LIN {X 0,Y 728.085,Z 811.922,A -85,B 0,C 180,E1 -1269.805,E2 -1269.805} C_VEL
LIN {X 0,Y 728.177,Z 799.737,A -85,B 0,C 180,E1 -1271.003,E2 -1271.003} C_VEL
LIN {X 0,Y 728.297,Z 785.992,A -85,B 0,C 180,E1 -1272.126,E2 -1272.126} C_VEL
LIN {X 0,Y 728.304,Z 784.724,A -85,B 0,C 180,E1 -1272.218,E2 -1272.218} C_VEL
LIN {X 0,Y 727.372,Z 779.122,A -85,B 0,C 180,E1 -1272.633,E2 -1272.633} C_VEL
LIN {X 0,Y 721.623,Z 764.762,A -85,B 0,C 180,E1 -1273.647,E2 -1273.647} C_VEL
LIN {X 0,Y 720.732,Z 758.498,A -85,B 0,C 180,E1 -1274.013,E2 -1274.013} C_VEL
LIN {X 0,Y 720.903,Z 741.804,A -85,B 0,C 180,E1 -1274.819,E2 -1274.819} C_VEL
LIN {X 0,Y 721.108,Z 724.487,A -85,B 0,C 180,E1 -1275.487,E2 -1275.487} C_VEL
LIN {X 0,Y 721.275,Z 705.803,A -85,B 0,C 180,E1 -1276.04,E2 -1276.04} C_VEL
LIN {X 0,Y 721.401,Z 686.903,A -85,B 0,C 180,E1 -1276.439,E2 -1276.439} C_VEL
LIN {X 0,Y 721.479,Z 666.781,A -85,B 0,C 180,E1 -1276.704,E2 -1276.704} C_VEL
LIN {X 0,Y 721.671,Z 473.025,A -85,B 0,C 180,E1 -1278.681,E2 -1278.681} C_VEL
LIN {X 0,Y 721.309,Z 469.724,A -85,B 0,C 180,E1 -1278.739,E2 -1278.739} C_VEL
LIN {X 0,Y 721.774,Z 418.133,A -85,B 0,C 180,E1 -1281.452,E2 -1281.452} C_VEL
LIN {X 0,Y 722.276,Z 363.537,A -85,B 0,C 180,E1 -1284.368,E2 -1284.368} C_VEL
LIN {X 0,Y 722.825,Z 311.685,A -85,B 0,C 180,E1 -1287.193,E2 -1287.193} C_VEL
LIN {X 0,Y 723.408,Z 258.979,A -85,B 0,C 180,E1 -1290.115,E2 -1290.115} C_VEL
LIN {X 0,Y 724.003,Z 208.72,A -85,B 0,C 180,E1 -1292.966,E2 -1292.966} C_VEL
LIN {X 0,Y 723.758,Z 205.468,A -85,B 0,C 180,E1 -1293.167,E2 -1293.167} C_VEL
LIN {X 0,Y 720.196,Z 195.523,A -85,B 0,C 180,E1 -1293.95,E2 -1293.95} C_VEL
LIN {X 0,Y 720.182,Z 195.518,A -85,B 0,C 180,E1 -1296.755,E2 -1296.755} C_VEL
LIN {X 0,Y 720.214,Z 195.521,A -85,B 0,C 180,E1 -1299.599,E2 -1299.599} C_VEL
LIN {X 0,Y 720.16,Z 195.522,A -85,B 0,C 180,E1 -1302.384,E2 -1302.384} C_VEL
LIN {X 0,Y 720.211,Z 195.516,A -85,B 0,C 180,E1 -1305.189,E2 -1305.189} C_VEL
LIN {X 0,Y 720.216,Z 195.521,A -85,B 0,C 180,E1 -1308.211,E2 -1308.211} C_VEL
LIN {X 0,Y 720.148,Z 195.522,A -85,B 0,C 180,E1 -1310.923,E2 -1310.923} C_VEL
LIN {X 0,Y 720.178,Z 195.522,A -85,B 0,C 180,E1 -1314.041,E2 -1314.041} C_VEL
LIN {X 0,Y 720.238,Z 195.651,A -85,B 0,C 180,E1 -1315.596,E2 -1315.596} C_VEL
LIN {X 0,Y 723.958,Z 206.616,A -85,B 0,C 180,E1 -1316.559,E2 -1316.559} C_VEL
LIN {X 0,Y 723.246,Z 247.825,A -85,B 0,C 180,E1 -1319.463,E2 -1319.463} C_VEL
LIN {X 0,Y 722.668,Z 288.727,A -85,B 0,C 180,E1 -1322.252,E2 -1322.252} C_VEL
LIN {X 0,Y 722.544,Z 304.623,A -85,B 0,C 180,E1 -1323.299,E2 -1323.299} C_VEL
LIN {X 0,Y 723.876,Z 312.314,A -85,B 0,C 180,E1 -1323.436,E2 -1323.436} C_VEL
LIN {X 0,Y 722.993,Z 604.896,A -85,B 0,C 180,E1 -1326.562,E2 -1326.562} C_VEL
LIN {X 0,Y 722.818,Z 626.619,A -85,B 0,C 180,E1 -1326.91,E2 -1326.91} C_VEL
LIN {X 0,Y 722.561,Z 650.13,A -85,B 0,C 180,E1 -1327.461,E2 -1327.461} C_VEL
LIN {X 0,Y 722.316,Z 669.51,A -85,B 0,C 180,E1 -1328.052,E2 -1328.052} C_VEL
LIN {X 0,Y 722.014,Z 689.697,A -85,B 0,C 180,E1 -1328.811,E2 -1328.811} C_VEL
LIN {X 0,Y 721.715,Z 710.059,A -85,B 0,C 180,E1 -1329.735,E2 -1329.735} C_VEL
LIN {X 0,Y 721.363,Z 729.936,A -85,B 0,C 180,E1 -1330.822,E2 -1330.822} C_VEL
LIN {X 0,Y 721.062,Z 746.81,A -85,B 0,C 180,E1 -1331.903,E2 -1331.903} C_VEL
LIN {X 0,Y 720.802,Z 763.918,A -85,B 0,C 180,E1 -1333.17,E2 -1333.17} C_VEL
LIN {X 0,Y 720.546,Z 779.819,A -85,B 0,C 180,E1 -1334.548,E2 -1334.548} C_VEL
LIN {X 0,Y 720.356,Z 792.902,A -85,B 0,C 180,E1 -1335.86,E2 -1335.86} C_VEL
LIN {X 0,Y 720.195,Z 806.207,A -85,B 0,C 180,E1 -1337.41,E2 -1337.41} C_VEL
LIN {X 0,Y 720.072,Z 817.974,A -85,B 0,C 180,E1 -1339.035,E2 -1339.035} C_VEL
LIN {X 0,Y 719.998,Z 827.271,A -85,B 0,C 180,E1 -1340.568,E2 -1340.568} C_VEL
LIN {X 0,Y 719.944,Z 835.631,A -85,B 0,C 180,E1 -1342.258,E2 -1342.258} C_VEL
LIN {X 0,Y 719.927,Z 842.505,A -85,B 0,C 180,E1 -1344.021,E2 -1344.021} C_VEL
LIN {X 0,Y 719.92,Z 847.512,A -85,B 0,C 180,E1 -1345.779,E2 -1345.779} C_VEL
LIN {X 0,Y 719.914,Z 850.607,A -85,B 0,C 180,E1 -1347.453,E2 -1347.453} C_VEL
LIN {X 0,Y 719.914,Z 852.289,A -85,B 0,C 180,E1 -1349.204,E2 -1349.204} C_VEL
LIN {X 0,Y 719.909,Z 852.219,A -85,B 0,C 180,E1 -1351.035,E2 -1351.035} C_VEL
LIN {X 0,Y 719.913,Z 850.51,A -85,B 0,C 180,E1 -1352.707,E2 -1352.707} C_VEL
LIN {X 0,Y 719.919,Z 847.147,A -85,B 0,C 180,E1 -1354.461,E2 -1354.461} C_VEL
LIN {X 0,Y 719.936,Z 841.735,A -85,B 0,C 180,E1 -1356.299,E2 -1356.299} C_VEL
LIN {X 0,Y 719.958,Z 834.828,A -85,B 0,C 180,E1 -1358.015,E2 -1358.015} C_VEL
LIN {X 0,Y 720.007,Z 826.408,A -85,B 0,C 180,E1 -1359.674,E2 -1359.674} C_VEL
LIN {X 0,Y 720.103,Z 815.862,A -85,B 0,C 180,E1 -1361.372,E2 -1361.372} C_VEL
LIN {X 0,Y 720.228,Z 804.11,A -85,B 0,C 180,E1 -1362.944,E2 -1362.944} C_VEL
LIN {X 0,Y 720.377,Z 791.433,A -85,B 0,C 180,E1 -1364.386,E2 -1364.386} C_VEL
LIN {X 0,Y 720.595,Z 776.326,A -85,B 0,C 180,E1 -1365.864,E2 -1365.864} C_VEL
LIN {X 0,Y 720.851,Z 759.998,A -85,B 0,C 180,E1 -1367.226,E2 -1367.226} C_VEL
LIN {X 0,Y 721.109,Z 744.471,A -85,B 0,C 180,E1 -1368.346,E2 -1368.346} C_VEL
LIN {X 0,Y 721.411,Z 726.463,A -85,B 0,C 180,E1 -1369.471,E2 -1369.471} C_VEL
LIN {X 0,Y 721.75,Z 706.47,A -85,B 0,C 180,E1 -1370.526,E2 -1370.526} C_VEL
LIN {X 0,Y 722.033,Z 688.563,A -85,B 0,C 180,E1 -1371.325,E2 -1371.325} C_VEL
LIN {X 0,Y 722.331,Z 668.395,A -85,B 0,C 180,E1 -1372.075,E2 -1372.075} C_VEL
LIN {X 0,Y 722.629,Z 645.716,A -85,B 0,C 180,E1 -1372.746,E2 -1372.746} C_VEL
LIN {X 0,Y 722.835,Z 624.224,A -85,B 0,C 180,E1 -1373.224,E2 -1373.224} C_VEL
LIN {X 0,Y 723.001,Z 603.601,A -85,B 0,C 180,E1 -1373.545,E2 -1373.545} C_VEL
LIN {X 0,Y 723.876,Z 312.433,A -85,B 0,C 180,E1 -1376.653,E2 -1376.653} C_VEL
LIN {X 0,Y 722.906,Z 306.324,A -85,B 0,C 180,E1 -1376.758,E2 -1376.758} C_VEL
LIN {X 0,Y 722.485,Z 303.913,A -85,B 0,C 180,E1 -1376.819,E2 -1376.819} C_VEL
LIN {X 0,Y 723.04,Z 261.674,A -85,B 0,C 180,E1 -1379.675,E2 -1379.675} C_VEL
LIN {X 0,Y 723.666,Z 220.838,A -85,B 0,C 180,E1 -1382.512,E2 -1382.512} C_VEL
LIN {X 0,Y 723.746,Z 206.018,A -85,B 0,C 180,E1 -1383.584,E2 -1383.584} C_VEL
LIN {X 0,Y 720.207,Z 195.519,A -85,B 0,C 180,E1 -1384.527,E2 -1384.527} C_VEL
LIN {X 0,Y 720.201,Z 195.524,A -85,B 0,C 180,E1 -1387.452,E2 -1387.452} C_VEL
LIN {X 0,Y 720.212,Z 195.511,A -85,B 0,C 180,E1 -1390.522,E2 -1390.522} C_VEL
LIN {X 0,Y 720.206,Z 195.521,A -85,B 0,C 180,E1 -1393.521,E2 -1393.521} C_VEL
LIN {X 0,Y 720.215,Z 195.509,A -85,B 0,C 180,E1 -1396.589,E2 -1396.589} C_VEL
LIN {X 0,Y 720.219,Z 195.519,A -85,B 0,C 180,E1 -1399.657,E2 -1399.657} C_VEL
LIN {X 0,Y 720.208,Z 195.509,A -85,B 0,C 180,E1 -1402.748,E2 -1402.748} C_VEL
LIN {X 0,Y 720.216,Z 195.521,A -85,B 0,C 180,E1 -1405.695,E2 -1405.695} C_VEL
LIN {X 0,Y 720.211,Z 195.51,A -85,B 0,C 180,E1 -1408.783,E2 -1408.783} C_VEL
LIN {X 0,Y 720.217,Z 195.517,A -85,B 0,C 180,E1 -1411.834,E2 -1411.834} C_VEL
LIN {X 0,Y 720.211,Z 195.51,A -85,B 0,C 180,E1 -1414.86,E2 -1414.86} C_VEL
LIN {X 0,Y 720.212,Z 195.52,A -85,B 0,C 180,E1 -1417.899,E2 -1417.899} C_VEL
LIN {X 0,Y 720.215,Z 195.507,A -85,B 0,C 180,E1 -1420.874,E2 -1420.874} C_VEL
LIN {X 0,Y 720.214,Z 195.52,A -85,B 0,C 180,E1 -1423.888,E2 -1423.888} C_VEL
LIN {X 0,Y 720.219,Z 195.506,A -85,B 0,C 180,E1 -1426.921,E2 -1426.921} C_VEL
LIN {X 0,Y 720.212,Z 195.52,A -85,B 0,C 180,E1 -1429.925,E2 -1429.925} C_VEL
LIN {X 0,Y 720.222,Z 195.506,A -85,B 0,C 180,E1 -1432.902,E2 -1432.902} C_VEL
LIN {X 0,Y 720.211,Z 195.521,A -85,B 0,C 180,E1 -1435.94,E2 -1435.94} C_VEL
LIN {X 0,Y 720.219,Z 195.508,A -85,B 0,C 180,E1 -1438.966,E2 -1438.966} C_VEL
LIN {X 0,Y 720.207,Z 195.52,A -85,B 0,C 180,E1 -1441.989,E2 -1441.989} C_VEL
LIN {X 0,Y 720.21,Z 195.51,A -85,B 0,C 180,E1 -1444.938,E2 -1444.938} C_VEL
LIN {X 0,Y 720.201,Z 195.518,A -85,B 0,C 180,E1 -1448.061,E2 -1448.061} C_VEL
LIN {X 0,Y 720.214,Z 195.51,A -85,B 0,C 180,E1 -1451.046,E2 -1451.046} C_VEL
LIN {X 0,Y 720.202,Z 195.52,A -85,B 0,C 180,E1 -1454.061,E2 -1454.061} C_VEL
LIN {X 0,Y 720.196,Z 195.512,A -85,B 0,C 180,E1 -1456.951,E2 -1456.951} C_VEL
LIN {X 0,Y 720.203,Z 195.521,A -85,B 0,C 180,E1 -1460.055,E2 -1460.055} C_VEL
LIN {X 0,Y 720.184,Z 195.514,A -85,B 0,C 180,E1 -1462.877,E2 -1462.877} C_VEL
LIN {X 0,Y 720.218,Z 195.522,A -85,B 0,C 180,E1 -1465.891,E2 -1465.891} C_VEL
LIN {X 0,Y 720.171,Z 195.516,A -85,B 0,C 180,E1 -1468.711,E2 -1468.711} C_VEL
LIN {X 0,Y 720.219,Z 195.515,A -85,B 0,C 180,E1 -1471.56,E2 -1471.56} C_VEL
LIN {X 0,Y 720.171,Z 195.519,A -85,B 0,C 180,E1 -1474.441,E2 -1474.441} C_VEL
LIN {X 0,Y 720.191,Z 195.514,A -85,B 0,C 180,E1 -1477.163,E2 -1477.163} C_VEL
LIN {X 0,Y 720.188,Z 195.522,A -85,B 0,C 180,E1 -1480.217,E2 -1480.217} C_VEL
LIN {X 0,Y 720.163,Z 195.518,A -85,B 0,C 180,E1 -1482.869,E2 -1482.869} C_VEL
LIN {X 0,Y 720.222,Z 195.518,A -85,B 0,C 180,E1 -1485.756,E2 -1485.756} C_VEL
LIN {X 0,Y 720.158,Z 195.522,A -85,B 0,C 180,E1 -1488.632,E2 -1488.632} C_VEL
LIN {X 0,Y 720.209,Z 195.663,A -85,B 0,C 180,E1 -1490.207,E2 -1490.207} C_VEL
LIN {X 0,Y 721.281,Z 198.701,A -85,B 0,C 180,E1 -1490.423,E2 -1490.423} C_VEL
LIN {X 0,Y 726.57,Z 209.646,A -85,B 0,C 180,E1 -1491.288,E2 -1491.288} C_VEL
LIN {X 0,Y 725.859,Z 260.94,A -85,B 0,C 180,E1 -1493.677,E2 -1493.677} C_VEL
LIN {X 0,Y 725.458,Z 299.229,A -85,B 0,C 180,E1 -1495.402,E2 -1495.402} C_VEL
LIN {X 0,Y 726.47,Z 307.17,A -85,B 0,C 180,E1 -1495.55,E2 -1495.55} C_VEL
LIN {X 0,Y 725.424,Z 570.263,A -85,B 0,C 180,E1 -1498.535,E2 -1498.535} C_VEL
LIN {X 0,Y 724.936,Z 690.96,A -85,B 0,C 180,E1 -1499.899,E2 -1499.899} C_VEL
LIN {X 0,Y 724.634,Z 716.508,A -85,B 0,C 180,E1 -1500.332,E2 -1500.332} C_VEL
LIN {X 0,Y 724.35,Z 738.123,A -85,B 0,C 180,E1 -1500.832,E2 -1500.832} C_VEL
LIN {X 0,Y 724.01,Z 761.286,A -85,B 0,C 180,E1 -1501.501,E2 -1501.501} C_VEL
LIN {X 0,Y 723.566,Z 783.363,A -85,B 0,C 180,E1 -1502.289,E2 -1502.289} C_VEL
LIN {X 0,Y 723.176,Z 805.236,A -85,B 0,C 180,E1 -1503.209,E2 -1503.209} C_VEL
LIN {X 0,Y 722.679,Z 827.148,A -85,B 0,C 180,E1 -1504.294,E2 -1504.294} C_VEL
LIN {X 0,Y 722.248,Z 847.62,A -85,B 0,C 180,E1 -1505.46,E2 -1505.46} C_VEL
LIN {X 0,Y 721.793,Z 867.842,A -85,B 0,C 180,E1 -1506.789,E2 -1506.789} C_VEL
LIN {X 0,Y 721.414,Z 886.71,A -85,B 0,C 180,E1 -1508.195,E2 -1508.195} C_VEL
LIN {X 0,Y 721.029,Z 904.462,A -85,B 0,C 180,E1 -1509.715,E2 -1509.715} C_VEL
LIN {X 0,Y 720.755,Z 920.964,A -85,B 0,C 180,E1 -1511.309,E2 -1511.309} C_VEL
LIN {X 0,Y 720.478,Z 935.22,A -85,B 0,C 180,E1 -1512.889,E2 -1512.889} C_VEL
LIN {X 0,Y 720.304,Z 948.442,A -85,B 0,C 180,E1 -1514.542,E2 -1514.542} C_VEL
LIN {X 0,Y 720.157,Z 960.276,A -85,B 0,C 180,E1 -1516.266,E2 -1516.266} C_VEL
LIN {X 0,Y 720.066,Z 970.03,A -85,B 0,C 180,E1 -1517.896,E2 -1517.896} C_VEL
LIN {X 0,Y 719.982,Z 980.182,A -85,B 0,C 180,E1 -1519.922,E2 -1519.922} C_VEL
LIN {X 0,Y 719.928,Z 986.815,A -85,B 0,C 180,E1 -1521.534,E2 -1521.534} C_VEL
LIN {X 0,Y 719.913,Z 993.245,A -85,B 0,C 180,E1 -1523.46,E2 -1523.46} C_VEL
LIN {X 0,Y 719.916,Z 997.813,A -85,B 0,C 180,E1 -1525.38,E2 -1525.38} C_VEL
LIN {X 0,Y 719.882,Z 1000.685,A -85,B 0,C 180,E1 -1527.134,E2 -1527.134} C_VEL
LIN {X 0,Y 719.891,Z 1002.262,A -85,B 0,C 180,E1 -1529.125,E2 -1529.125} C_VEL
LIN {X 0,Y 719.883,Z 1002.306,A -85,B 0,C 180,E1 -1530.716,E2 -1530.716} C_VEL
LIN {X 0,Y 719.888,Z 1001.017,A -85,B 0,C 180,E1 -1532.627,E2 -1532.627} C_VEL
LIN {X 0,Y 719.917,Z 997.971,A -85,B 0,C 180,E1 -1534.541,E2 -1534.541} C_VEL
LIN {X 0,Y 719.915,Z 993.864,A -85,B 0,C 180,E1 -1536.299,E2 -1536.299} C_VEL
LIN {X 0,Y 719.936,Z 987.422,A -85,B 0,C 180,E1 -1538.305,E2 -1538.305} C_VEL
LIN {X 0,Y 719.968,Z 980.892,A -85,B 0,C 180,E1 -1539.916,E2 -1539.916} C_VEL
LIN {X 0,Y 720.053,Z 971.867,A -85,B 0,C 180,E1 -1541.779,E2 -1541.779} C_VEL
LIN {X 0,Y 720.143,Z 961.081,A -85,B 0,C 180,E1 -1543.608,E2 -1543.608} C_VEL
LIN {X 0,Y 720.295,Z 949.06,A -85,B 0,C 180,E1 -1545.375,E2 -1545.375} C_VEL
LIN {X 0,Y 720.472,Z 935.927,A -85,B 0,C 180,E1 -1547.028,E2 -1547.028} C_VEL
LIN {X 0,Y 720.739,Z 921.74,A -85,B 0,C 180,E1 -1548.607,E2 -1548.607} C_VEL
LIN {X 0,Y 721.008,Z 905.39,A -85,B 0,C 180,E1 -1550.201,E2 -1550.201} C_VEL
LIN {X 0,Y 721.376,Z 888.27,A -85,B 0,C 180,E1 -1551.678,E2 -1551.678} C_VEL
LIN {X 0,Y 721.76,Z 869.107,A -85,B 0,C 180,E1 -1553.121,E2 -1553.121} C_VEL
LIN {X 0,Y 722.231,Z 849.066,A -85,B 0,C 180,E1 -1554.453,E2 -1554.453} C_VEL
LIN {X 0,Y 722.653,Z 827.944,A -85,B 0,C 180,E1 -1555.663,E2 -1555.663} C_VEL
LIN {X 0,Y 723.165,Z 806.229,A -85,B 0,C 180,E1 -1556.747,E2 -1556.747} C_VEL
LIN {X 0,Y 723.547,Z 784.481,A -85,B 0,C 180,E1 -1557.667,E2 -1557.667} C_VEL
LIN {X 0,Y 723.972,Z 762.568,A -85,B 0,C 180,E1 -1558.456,E2 -1558.456} C_VEL
LIN {X 0,Y 724.349,Z 738.334,A -85,B 0,C 180,E1 -1559.162,E2 -1559.162} C_VEL
LIN {X 0,Y 724.63,Z 716.764,A -85,B 0,C 180,E1 -1559.663,E2 -1559.663} C_VEL
LIN {X 0,Y 724.936,Z 691.166,A -85,B 0,C 180,E1 -1560.098,E2 -1560.098} C_VEL
LIN {X 0,Y 725.376,Z 582.637,A -85,B 0,C 180,E1 -1561.326,E2 -1561.326} C_VEL
LIN {X 0,Y 726.451,Z 311.994,A -85,B 0,C 180,E1 -1564.394,E2 -1564.394} C_VEL
LIN {X 0,Y 726.227,Z 304.001,A -85,B 0,C 180,E1 -1564.5,E2 -1564.5} C_VEL
LIN {X 0,Y 725.36,Z 298.429,A -85,B 0,C 180,E1 -1564.618,E2 -1564.618} C_VEL
LIN {X 0,Y 726.223,Z 237.623,A -85,B 0,C 180,E1 -1567.398,E2 -1567.398} C_VEL
LIN {X 0,Y 726.566,Z 209.659,A -85,B 0,C 180,E1 -1568.712,E2 -1568.712} C_VEL
LIN {X 0,Y 721.385,Z 198.876,A -85,B 0,C 180,E1 -1569.587,E2 -1569.587} C_VEL
LIN {X 0,Y 720.172,Z 195.526,A -85,B 0,C 180,E1 -1569.844,E2 -1569.844} C_VEL
LIN {X 0,Y 720.211,Z 195.521,A -85,B 0,C 180,E1 -1572.858,E2 -1572.858} C_VEL
LIN {X 0,Y 720.177,Z 195.524,A -85,B 0,C 180,E1 -1575.704,E2 -1575.704} C_VEL
LIN {X 0,Y 720.221,Z 195.519,A -85,B 0,C 180,E1 -1578.684,E2 -1578.684} C_VEL
LIN {X 0,Y 720.195,Z 195.524,A -85,B 0,C 180,E1 -1581.668,E2 -1581.668} C_VEL
LIN {X 0,Y 720.223,Z 195.521,A -85,B 0,C 180,E1 -1584.625,E2 -1584.625} C_VEL
LIN {X 0,Y 720.201,Z 195.528,A -85,B 0,C 180,E1 -1586.094,E2 -1586.094} C_VEL
LIN {X 0,Y 724.343,Z 207.121,A -85,B 0,C 180,E1 -1587.052,E2 -1587.052} C_VEL
LIN {X 0,Y 723.304,Z 257.17,A -85,B 0,C 180,E1 -1589.926,E2 -1589.926} C_VEL
LIN {X 0,Y 722.6,Z 315.269,A -85,B 0,C 180,E1 -1593.141,E2 -1593.141} C_VEL
LIN {X 0,Y 722.176,Z 369.58,A -85,B 0,C 180,E1 -1596.067,E2 -1596.067} C_VEL
LIN {X 0,Y 721.73,Z 424.416,A -85,B 0,C 180,E1 -1598.972,E2 -1598.972} C_VEL
LIN {X 0,Y 721.364,Z 470.562,A -85,B 0,C 180,E1 -1601.375,E2 -1601.375} C_VEL
LIN {X 0,Y 721.822,Z 478.064,A -85,B 0,C 180,E1 -1601.465,E2 -1601.465} C_VEL
LIN {X 0,Y 721.438,Z 679.938,A -85,B 0,C 180,E1 -1603.541,E2 -1603.541} C_VEL
LIN {X 0,Y 721.316,Z 699.052,A -85,B 0,C 180,E1 -1603.89,E2 -1603.89} C_VEL
LIN {X 0,Y 721.167,Z 717.241,A -85,B 0,C 180,E1 -1604.371,E2 -1604.371} C_VEL
LIN {X 0,Y 720.969,Z 734.998,A -85,B 0,C 180,E1 -1604.992,E2 -1604.992} C_VEL
LIN {X 0,Y 720.803,Z 751.994,A -85,B 0,C 180,E1 -1605.746,E2 -1605.746} C_VEL
LIN {X 0,Y 720.617,Z 767.716,A -85,B 0,C 180,E1 -1606.602,E2 -1606.602} C_VEL
LIN {X 0,Y 720.432,Z 783.102,A -85,B 0,C 180,E1 -1607.618,E2 -1607.618} C_VEL
LIN {X 0,Y 720.274,Z 796.852,A -85,B 0,C 180,E1 -1608.712,E2 -1608.712} C_VEL
LIN {X 0,Y 720.145,Z 809.523,A -85,B 0,C 180,E1 -1609.924,E2 -1609.924} C_VEL
LIN {X 0,Y 720.05,Z 820.643,A -85,B 0,C 180,E1 -1611.214,E2 -1611.214} C_VEL
LIN {X 0,Y 719.983,Z 830.232,A -85,B 0,C 180,E1 -1612.579,E2 -1612.579} C_VEL
LIN {X 0,Y 719.946,Z 837.854,A -85,B 0,C 180,E1 -1613.941,E2 -1613.941} C_VEL
LIN {X 0,Y 719.921,Z 844.045,A -85,B 0,C 180,E1 -1615.379,E2 -1615.379} C_VEL
LIN {X 0,Y 719.914,Z 848.466,A -85,B 0,C 180,E1 -1616.815,E2 -1616.815} C_VEL
LIN {X 0,Y 719.912,Z 851.34,A -85,B 0,C 180,E1 -1618.329,E2 -1618.329} C_VEL
LIN {X 0,Y 719.912,Z 852.449,A -85,B 0,C 180,E1 -1619.841,E2 -1619.841} C_VEL
LIN {X 0,Y 719.913,Z 851.819,A -85,B 0,C 180,E1 -1621.353,E2 -1621.353} C_VEL
LIN {X 0,Y 719.914,Z 849.435,A -85,B 0,C 180,E1 -1622.866,E2 -1622.866} C_VEL
LIN {X 0,Y 719.922,Z 845.232,A -85,B 0,C 180,E1 -1624.381,E2 -1624.381} C_VEL
LIN {X 0,Y 719.936,Z 839.461,A -85,B 0,C 180,E1 -1625.819,E2 -1625.819} C_VEL
LIN {X 0,Y 719.981,Z 831.802,A -85,B 0,C 180,E1 -1627.26,E2 -1627.26} C_VEL
LIN {X 0,Y 720.037,Z 822.605,A -85,B 0,C 180,E1 -1628.626,E2 -1628.626} C_VEL
LIN {X 0,Y 720.131,Z 811.918,A -85,B 0,C 180,E1 -1629.914,E2 -1629.914} C_VEL
LIN {X 0,Y 720.249,Z 799.731,A -85,B 0,C 180,E1 -1631.126,E2 -1631.126} C_VEL
LIN {X 0,Y 720.4,Z 785.987,A -85,B 0,C 180,E1 -1632.261,E2 -1632.261} C_VEL
LIN {X 0,Y 720.572,Z 771.146,A -85,B 0,C 180,E1 -1633.279,E2 -1633.279} C_VEL
LIN {X 0,Y 720.732,Z 758.498,A -85,B 0,C 180,E1 -1634.013,E2 -1634.013} C_VEL
LIN {X 0,Y 719.842,Z 752.168,A -85,B 0,C 180,E1 -1634.364,E2 -1634.364} C_VEL
LIN {X 0,Y 714.42,Z 736.944,A -85,B 0,C 180,E1 -1635.164,E2 -1635.164} C_VEL
LIN {X 0,Y 713.298,Z 730.158,A -85,B 0,C 180,E1 -1635.452,E2 -1635.452} C_VEL
LIN {X 0,Y 713.28,Z 729.152,A -85,B 0,C 180,E1 -1635.489,E2 -1635.489} C_VEL
LIN {X 0,Y 713.505,Z 710.535,A -85,B 0,C 180,E1 -1636.089,E2 -1636.089} C_VEL
LIN {X 0,Y 713.666,Z 691.674,A -85,B 0,C 180,E1 -1636.532,E2 -1636.532} C_VEL
LIN {X 0,Y 713.79,Z 672.625,A -85,B 0,C 180,E1 -1636.823,E2 -1636.823} C_VEL
LIN {X 0,Y 714.094,Z 473.867,A -85,B 0,C 180,E1 -1638.879,E2 -1638.879} C_VEL
LIN {X 0,Y 713.625,Z 469.588,A -85,B 0,C 180,E1 -1638.955,E2 -1638.955} C_VEL
LIN {X 0,Y 714.172,Z 418.046,A -85,B 0,C 180,E1 -1641.692,E2 -1641.692} C_VEL
LIN {X 0,Y 714.783,Z 362.685,A -85,B 0,C 180,E1 -1644.681,E2 -1644.681} C_VEL
LIN {X 0,Y 715.433,Z 312.1,A -85,B 0,C 180,E1 -1647.465,E2 -1647.465} C_VEL
LIN {X 0,Y 716.158,Z 259.687,A -85,B 0,C 180,E1 -1650.401,E2 -1650.401} C_VEL
LIN {X 0,Y 716.883,Z 210.15,A -85,B 0,C 180,E1 -1653.24,E2 -1653.24} C_VEL
LIN {X 0,Y 716.315,Z 207.723,A -85,B 0,C 180,E1 -1653.411,E2 -1653.411} C_VEL
LIN {X 0,Y 712.272,Z 196.512,A -85,B 0,C 180,E1 -1654.307,E2 -1654.307} C_VEL
LIN {X 0,Y 712.274,Z 196.504,A -85,B 0,C 180,E1 -1657.333,E2 -1657.333} C_VEL
LIN {X 0,Y 712.208,Z 196.513,A -85,B 0,C 180,E1 -1660.227,E2 -1660.227} C_VEL
LIN {X 0,Y 712.269,Z 196.511,A -85,B 0,C 180,E1 -1662.91,E2 -1662.91} C_VEL
LIN {X 0,Y 712.265,Z 196.505,A -85,B 0,C 180,E1 -1665.869,E2 -1665.869} C_VEL
LIN {X 0,Y 712.235,Z 196.508,A -85,B 0,C 180,E1 -1668.714,E2 -1668.714} C_VEL
LIN {X 0,Y 712.276,Z 196.512,A -85,B 0,C 180,E1 -1671.566,E2 -1671.566} C_VEL
LIN {X 0,Y 712.234,Z 196.514,A -85,B 0,C 180,E1 -1674.464,E2 -1674.464} C_VEL
LIN {X 0,Y 712.28,Z 196.515,A -85,B 0,C 180,E1 -1675.207,E2 -1675.207} C_VEL
LIN {X 0,Y 716.825,Z 210.095,A -85,B 0,C 180,E1 -1676.417,E2 -1676.417} C_VEL
LIN {X 0,Y 715.958,Z 248.509,A -85,B 0,C 180,E1 -1679.166,E2 -1679.166} C_VEL
LIN {X 0,Y 715.265,Z 289.395,A -85,B 0,C 180,E1 -1681.985,E2 -1681.985} C_VEL
LIN {X 0,Y 715.109,Z 304.617,A -85,B 0,C 180,E1 -1682.999,E2 -1682.999} C_VEL
LIN {X 0,Y 716.715,Z 313.568,A -85,B 0,C 180,E1 -1683.163,E2 -1683.163} C_VEL
LIN {X 0,Y 715.65,Z 604.587,A -85,B 0,C 180,E1 -1686.302,E2 -1686.302} C_VEL
LIN {X 0,Y 715.451,Z 625.147,A -85,B 0,C 180,E1 -1686.631,E2 -1686.631} C_VEL
LIN {X 0,Y 715.193,Z 647.921,A -85,B 0,C 180,E1 -1687.15,E2 -1687.15} C_VEL
LIN {X 0,Y 714.824,Z 669.791,A -85,B 0,C 180,E1 -1687.82,E2 -1687.82} C_VEL
LIN {X 0,Y 714.474,Z 689.691,A -85,B 0,C 180,E1 -1688.576,E2 -1688.576} C_VEL
LIN {X 0,Y 714.107,Z 710.089,A -85,B 0,C 180,E1 -1689.511,E2 -1689.511} C_VEL
LIN {X 0,Y 713.674,Z 729.931,A -85,B 0,C 180,E1 -1690.607,E2 -1690.607} C_VEL
LIN {X 0,Y 713.324,Z 746.817,A -85,B 0,C 180,E1 -1691.7,E2 -1691.7} C_VEL
LIN {X 0,Y 713.005,Z 763.646,A -85,B 0,C 180,E1 -1692.957,E2 -1692.957} C_VEL
LIN {X 0,Y 712.691,Z 779.818,A -85,B 0,C 180,E1 -1694.373,E2 -1694.373} C_VEL
LIN {X 0,Y 712.46,Z 792.9,A -85,B 0,C 180,E1 -1695.7,E2 -1695.7} C_VEL
LIN {X 0,Y 712.265,Z 806.215,A -85,B 0,C 180,E1 -1697.267,E2 -1697.267} C_VEL
LIN {X 0,Y 712.105,Z 818.482,A -85,B 0,C 180,E1 -1698.991,E2 -1698.991} C_VEL
LIN {X 0,Y 712.016,Z 827.705,A -85,B 0,C 180,E1 -1700.543,E2 -1700.543} C_VEL
LIN {X 0,Y 711.958,Z 835.635,A -85,B 0,C 180,E1 -1702.17,E2 -1702.17} C_VEL
LIN {X 0,Y 711.934,Z 842.509,A -85,B 0,C 180,E1 -1703.953,E2 -1703.953} C_VEL
LIN {X 0,Y 711.922,Z 847.507,A -85,B 0,C 180,E1 -1705.731,E2 -1705.731} C_VEL
LIN {X 0,Y 711.915,Z 850.608,A -85,B 0,C 180,E1 -1707.424,E2 -1707.424} C_VEL
LIN {X 0,Y 711.914,Z 852.292,A -85,B 0,C 180,E1 -1709.195,E2 -1709.195} C_VEL
LIN {X 0,Y 711.909,Z 852.214,A -85,B 0,C 180,E1 -1711.046,E2 -1711.046} C_VEL
LIN {X 0,Y 711.912,Z 850.509,A -85,B 0,C 180,E1 -1712.737,E2 -1712.737} C_VEL
LIN {X 0,Y 711.919,Z 847.149,A -85,B 0,C 180,E1 -1714.511,E2 -1714.511} C_VEL
LIN {X 0,Y 711.937,Z 841.731,A -85,B 0,C 180,E1 -1716.37,E2 -1716.37} C_VEL
LIN {X 0,Y 711.97,Z 834.967,A -85,B 0,C 180,E1 -1718.073,E2 -1718.073} C_VEL
LIN {X 0,Y 712.034,Z 826.408,A -85,B 0,C 180,E1 -1719.783,E2 -1719.783} C_VEL
LIN {X 0,Y 712.148,Z 815.858,A -85,B 0,C 180,E1 -1721.5,E2 -1721.5} C_VEL
LIN {X 0,Y 712.297,Z 804.33,A -85,B 0,C 180,E1 -1723.062,E2 -1723.062} C_VEL
LIN {X 0,Y 712.49,Z 791.429,A -85,B 0,C 180,E1 -1724.549,E2 -1724.549} C_VEL
LIN {X 0,Y 712.751,Z 776.122,A -85,B 0,C 180,E1 -1726.062,E2 -1726.062} C_VEL
LIN {X 0,Y 713.054,Z 760.059,A -85,B 0,C 180,E1 -1727.415,E2 -1727.415} C_VEL
LIN {X 0,Y 713.377,Z 744.454,A -85,B 0,C 180,E1 -1728.552,E2 -1728.552} C_VEL
LIN {X 0,Y 713.758,Z 726.057,A -85,B 0,C 180,E1 -1729.712,E2 -1729.712} C_VEL
LIN {X 0,Y 714.156,Z 705.733,A -85,B 0,C 180,E1 -1730.789,E2 -1730.789} C_VEL
LIN {X 0,Y 714.511,Z 687.71,A -85,B 0,C 180,E1 -1731.595,E2 -1731.595} C_VEL
LIN {X 0,Y 714.85,Z 668.384,A -85,B 0,C 180,E1 -1732.319,E2 -1732.319} C_VEL
LIN {X 0,Y 715.217,Z 645.269,A -85,B 0,C 180,E1 -1733.006,E2 -1733.006} C_VEL
LIN {X 0,Y 715.465,Z 624.006,A -85,B 0,C 180,E1 -1733.48,E2 -1733.48} C_VEL
LIN {X 0,Y 715.653,Z 604.059,A -85,B 0,C 180,E1 -1733.794,E2 -1733.794} C_VEL
LIN {X 0,Y 716.712,Z 314.22,A -85,B 0,C 180,E1 -1736.92,E2 -1736.92} C_VEL
LIN {X 0,Y 716.168,Z 309.757,A -85,B 0,C 180,E1 -1736.992,E2 -1736.992} C_VEL
LIN {X 0,Y 715.054,Z 303.905,A -85,B 0,C 180,E1 -1737.12,E2 -1737.12} C_VEL
LIN {X 0,Y 715.713,Z 262.054,A -85,B 0,C 180,E1 -1739.982,E2 -1739.982} C_VEL
LIN {X 0,Y 716.51,Z 225.81,A -85,B 0,C 180,E1 -1742.554,E2 -1742.554} C_VEL
LIN {X 0,Y 716.649,Z 209.27,A -85,B 0,C 180,E1 -1743.74,E2 -1743.74} C_VEL
LIN {X 0,Y 712.244,Z 196.513,A -85,B 0,C 180,E1 -1744.913,E2 -1744.913} C_VEL
LIN {X 0,Y 712.279,Z 196.512,A -85,B 0,C 180,E1 -1747.783,E2 -1747.783} C_VEL
LIN {X 0,Y 712.256,Z 196.503,A -85,B 0,C 180,E1 -1750.752,E2 -1750.752} C_VEL
LIN {X 0,Y 712.28,Z 196.508,A -85,B 0,C 180,E1 -1753.701,E2 -1753.701} C_VEL
LIN {X 0,Y 712.26,Z 196.5,A -85,B 0,C 180,E1 -1756.768,E2 -1756.768} C_VEL
LIN {X 0,Y 712.281,Z 196.507,A -85,B 0,C 180,E1 -1759.778,E2 -1759.778} C_VEL
LIN {X 0,Y 712.268,Z 196.498,A -85,B 0,C 180,E1 -1762.768,E2 -1762.768} C_VEL
LIN {X 0,Y 712.277,Z 196.508,A -85,B 0,C 180,E1 -1765.775,E2 -1765.775} C_VEL
LIN {X 0,Y 712.271,Z 196.5,A -85,B 0,C 180,E1 -1768.801,E2 -1768.801} C_VEL
LIN {X 0,Y 712.276,Z 196.506,A -85,B 0,C 180,E1 -1771.857,E2 -1771.857} C_VEL
LIN {X 0,Y 712.269,Z 196.499,A -85,B 0,C 180,E1 -1774.916,E2 -1774.916} C_VEL
LIN {X 0,Y 712.273,Z 196.509,A -85,B 0,C 180,E1 -1777.9,E2 -1777.9} C_VEL
LIN {X 0,Y 712.274,Z 196.496,A -85,B 0,C 180,E1 -1780.908,E2 -1780.908} C_VEL
LIN {X 0,Y 712.27,Z 196.508,A -85,B 0,C 180,E1 -1783.945,E2 -1783.945} C_VEL
LIN {X 0,Y 712.277,Z 196.495,A -85,B 0,C 180,E1 -1786.965,E2 -1786.965} C_VEL
LIN {X 0,Y 712.268,Z 196.509,A -85,B 0,C 180,E1 -1789.975,E2 -1789.975} C_VEL
LIN {X 0,Y 712.279,Z 196.496,A -85,B 0,C 180,E1 -1792.985,E2 -1792.985} C_VEL
LIN {X 0,Y 712.263,Z 196.508,A -85,B 0,C 180,E1 -1796.056,E2 -1796.056} C_VEL
LIN {X 0,Y 712.282,Z 196.497,A -85,B 0,C 180,E1 -1799.035,E2 -1799.035} C_VEL
LIN {X 0,Y 712.26,Z 196.507,A -85,B 0,C 180,E1 -1802.092,E2 -1802.092} C_VEL
LIN {X 0,Y 712.278,Z 196.499,A -85,B 0,C 180,E1 -1805.074,E2 -1805.074} C_VEL
LIN {X 0,Y 712.262,Z 196.507,A -85,B 0,C 180,E1 -1808.07,E2 -1808.07} C_VEL
LIN {X 0,Y 712.271,Z 196.5,A -85,B 0,C 180,E1 -1811.006,E2 -1811.006} C_VEL
LIN {X 0,Y 712.263,Z 196.509,A -85,B 0,C 180,E1 -1814.06,E2 -1814.06} C_VEL
LIN {X 0,Y 712.261,Z 196.501,A -85,B 0,C 180,E1 -1816.978,E2 -1816.978} C_VEL
LIN {X 0,Y 712.258,Z 196.509,A -85,B 0,C 180,E1 -1820.117,E2 -1820.117} C_VEL
LIN {X 0,Y 712.252,Z 196.503,A -85,B 0,C 180,E1 -1822.971,E2 -1822.971} C_VEL
LIN {X 0,Y 712.265,Z 196.508,A -85,B 0,C 180,E1 -1826.065,E2 -1826.065} C_VEL
LIN {X 0,Y 712.238,Z 196.503,A -85,B 0,C 180,E1 -1828.877,E2 -1828.877} C_VEL
LIN {X 0,Y 712.281,Z 196.508,A -85,B 0,C 180,E1 -1831.865,E2 -1831.865} C_VEL
LIN {X 0,Y 712.228,Z 196.507,A -85,B 0,C 180,E1 -1834.651,E2 -1834.651} C_VEL
LIN {X 0,Y 712.281,Z 196.504,A -85,B 0,C 180,E1 -1837.52,E2 -1837.52} C_VEL
LIN {X 0,Y 712.23,Z 196.51,A -85,B 0,C 180,E1 -1840.456,E2 -1840.456} C_VEL
LIN {X 0,Y 712.251,Z 196.505,A -85,B 0,C 180,E1 -1843.231,E2 -1843.231} C_VEL
LIN {X 0,Y 712.24,Z 196.514,A -85,B 0,C 180,E1 -1846.314,E2 -1846.314} C_VEL
LIN {X 0,Y 712.22,Z 196.51,A -85,B 0,C 180,E1 -1848.929,E2 -1848.929} C_VEL
LIN {X 0,Y 712.307,Z 196.683,A -85,B 0,C 180,E1 -1849.741,E2 -1849.741} C_VEL
LIN {X 0,Y 713.368,Z 199.645,A -85,B 0,C 180,E1 -1849.957,E2 -1849.957} C_VEL
LIN {X 0,Y 719.946,Z 213.509,A -85,B 0,C 180,E1 -1851.055,E2 -1851.055} C_VEL
LIN {X 0,Y 719.057,Z 267.233,A -85,B 0,C 180,E1 -1853.575,E2 -1853.575} C_VEL
LIN {X 0,Y 718.641,Z 299.284,A -85,B 0,C 180,E1 -1855.027,E2 -1855.027} C_VEL
LIN {X 0,Y 719.861,Z 308.443,A -85,B 0,C 180,E1 -1855.203,E2 -1855.203} C_VEL
LIN {X 0,Y 718.584,Z 572.549,A -85,B 0,C 180,E1 -1858.227,E2 -1858.227} C_VEL
LIN {X 0,Y 718.004,Z 691.175,A -85,B 0,C 180,E1 -1859.581,E2 -1859.581} C_VEL
LIN {X 0,Y 717.648,Z 716.767,A -85,B 0,C 180,E1 -1860.019,E2 -1860.019} C_VEL
LIN {X 0,Y 717.298,Z 738.46,A -85,B 0,C 180,E1 -1860.526,E2 -1860.526} C_VEL
LIN {X 0,Y 716.853,Z 762.568,A -85,B 0,C 180,E1 -1861.235,E2 -1861.235} C_VEL
LIN {X 0,Y 716.339,Z 784.486,A -85,B 0,C 180,E1 -1862.031,E2 -1862.031} C_VEL
LIN {X 0,Y 715.831,Z 807.582,A -85,B 0,C 180,E1 -1863.022,E2 -1863.022} C_VEL
LIN {X 0,Y 715.246,Z 828.756,A -85,B 0,C 180,E1 -1864.096,E2 -1864.096} C_VEL
LIN {X 0,Y 714.719,Z 849.755,A -85,B 0,C 180,E1 -1865.317,E2 -1865.317} C_VEL
LIN {X 0,Y 714.182,Z 869.143,A -85,B 0,C 180,E1 -1866.621,E2 -1866.621} C_VEL
LIN {X 0,Y 713.72,Z 887.819,A -85,B 0,C 180,E1 -1868.039,E2 -1868.039} C_VEL
LIN {X 0,Y 713.298,Z 904.462,A -85,B 0,C 180,E1 -1869.485,E2 -1869.485} C_VEL
LIN {X 0,Y 712.937,Z 920.965,A -85,B 0,C 180,E1 -1871.096,E2 -1871.096} C_VEL
LIN {X 0,Y 712.616,Z 935.222,A -85,B 0,C 180,E1 -1872.695,E2 -1872.695} C_VEL
LIN {X 0,Y 712.389,Z 949.06,A -85,B 0,C 180,E1 -1874.45,E2 -1874.45} C_VEL
LIN {X 0,Y 712.21,Z 960.797,A -85,B 0,C 180,E1 -1876.192,E2 -1876.192} C_VEL
LIN {X 0,Y 712.093,Z 970.948,A -85,B 0,C 180,E1 -1877.923,E2 -1877.923} C_VEL
LIN {X 0,Y 711.997,Z 980.538,A -85,B 0,C 180,E1 -1879.89,E2 -1879.89} C_VEL
LIN {X 0,Y 711.935,Z 987.12,A -85,B 0,C 180,E1 -1881.52,E2 -1881.52} C_VEL
LIN {X 0,Y 711.916,Z 993.451,A -85,B 0,C 180,E1 -1883.468,E2 -1883.468} C_VEL
LIN {X 0,Y 711.913,Z 997.814,A -85,B 0,C 180,E1 -1885.327,E2 -1885.327} C_VEL
LIN {X 0,Y 711.882,Z 1000.685,A -85,B 0,C 180,E1 -1887.102,E2 -1887.102} C_VEL
LIN {X 0,Y 711.891,Z 1002.262,A -85,B 0,C 180,E1 -1889.115,E2 -1889.115} C_VEL
LIN {X 0,Y 711.883,Z 1002.306,A -85,B 0,C 180,E1 -1890.724,E2 -1890.724} C_VEL
LIN {X 0,Y 711.887,Z 1001.017,A -85,B 0,C 180,E1 -1892.657,E2 -1892.657} C_VEL
LIN {X 0,Y 711.917,Z 997.972,A -85,B 0,C 180,E1 -1894.592,E2 -1894.592} C_VEL
LIN {X 0,Y 711.915,Z 993.864,A -85,B 0,C 180,E1 -1896.37,E2 -1896.37} C_VEL
LIN {X 0,Y 711.937,Z 987.423,A -85,B 0,C 180,E1 -1898.399,E2 -1898.399} C_VEL
LIN {X 0,Y 711.989,Z 980.892,A -85,B 0,C 180,E1 -1900.029,E2 -1900.029} C_VEL
LIN {X 0,Y 712.085,Z 971.866,A -85,B 0,C 180,E1 -1901.912,E2 -1901.912} C_VEL
LIN {X 0,Y 712.2,Z 961.318,A -85,B 0,C 180,E1 -1903.725,E2 -1903.725} C_VEL
LIN {X 0,Y 712.375,Z 949.642,A -85,B 0,C 180,E1 -1905.467,E2 -1905.467} C_VEL
LIN {X 0,Y 712.602,Z 935.929,A -85,B 0,C 180,E1 -1907.222,E2 -1907.222} C_VEL
LIN {X 0,Y 712.922,Z 921.741,A -85,B 0,C 180,E1 -1908.819,E2 -1908.819} C_VEL
LIN {X 0,Y 713.27,Z 905.39,A -85,B 0,C 180,E1 -1910.43,E2 -1910.43} C_VEL
LIN {X 0,Y 713.688,Z 888.776,A -85,B 0,C 180,E1 -1911.881,E2 -1911.881} C_VEL
LIN {X 0,Y 714.166,Z 869.652,A -85,B 0,C 180,E1 -1913.342,E2 -1913.342} C_VEL
LIN {X 0,Y 714.698,Z 850.418,A -85,B 0,C 180,E1 -1914.64,E2 -1914.64} C_VEL
LIN {X 0,Y 715.218,Z 829.552,A -85,B 0,C 180,E1 -1915.861,E2 -1915.861} C_VEL
LIN {X 0,Y 715.786,Z 808.975,A -85,B 0,C 180,E1 -1916.911,E2 -1916.911} C_VEL
LIN {X 0,Y 716.313,Z 785.727,A -85,B 0,C 180,E1 -1917.92,E2 -1917.92} C_VEL
LIN {X 0,Y 716.771,Z 765.133,A -85,B 0,C 180,E1 -1918.678,E2 -1918.678} C_VEL
LIN {X 0,Y 717.283,Z 740.116,A -85,B 0,C 180,E1 -1919.43,E2 -1919.43} C_VEL
LIN {X 0,Y 717.613,Z 718.69,A -85,B 0,C 180,E1 -1919.94,E2 -1919.94} C_VEL
LIN {X 0,Y 717.992,Z 693.629,A -85,B 0,C 180,E1 -1920.386,E2 -1920.386} C_VEL
LIN {X 0,Y 718.269,Z 642.02,A -85,B 0,C 180,E1 -1920.991,E2 -1920.991} C_VEL
LIN {X 0,Y 719.445,Z 392.284,A -85,B 0,C 180,E1 -1923.827,E2 -1923.827} C_VEL
LIN {X 0,Y 719.68,Z 305.755,A -85,B 0,C 180,E1 -1924.839,E2 -1924.839} C_VEL
LIN {X 0,Y 718.539,Z 298.171,A -85,B 0,C 180,E1 -1925.007,E2 -1925.007} C_VEL
LIN {X 0,Y 719.603,Z 236.709,A -85,B 0,C 180,E1 -1927.846,E2 -1927.846} C_VEL
LIN {X 0,Y 719.965,Z 213.374,A -85,B 0,C 180,E1 -1928.946,E2 -1928.946} C_VEL
LIN {X 0,Y 713.431,Z 199.808,A -85,B 0,C 180,E1 -1930.072,E2 -1930.072} C_VEL
LIN {X 0,Y 712.281,Z 196.511,A -85,B 0,C 180,E1 -1930.336,E2 -1930.336} C_VEL
LIN {X 0,Y 712.279,Z 196.511,A -85,B 0,C 180,E1 -1933.24,E2 -1933.24} C_VEL
LIN {X 0,Y 712.282,Z 196.51,A -85,B 0,C 180,E1 -1936.206,E2 -1936.206} C_VEL
LIN {X 0,Y 712.264,Z 196.512,A -85,B 0,C 180,E1 -1939.171,E2 -1939.171} C_VEL
LIN {X 0,Y 712.28,Z 196.51,A -85,B 0,C 180,E1 -1942.086,E2 -1942.086} C_VEL
LIN {X 0,Y 712.252,Z 196.514,A -85,B 0,C 180,E1 -1945.069,E2 -1945.069} C_VEL
LIN {X 0,Y 712.253,Z 196.683,A -85,B 0,C 180,E1 -1945.655,E2 -1945.655} C_VEL
LIN {X 0,Y 717.389,Z 210.124,A -85,B 0,C 180,E1 -1946.834,E2 -1946.834} C_VEL
LIN {X 0,Y 716.102,Z 258.891,A -85,B 0,C 180,E1 -1949.684,E2 -1949.684} C_VEL
LIN {X 0,Y 715.192,Z 315.897,A -85,B 0,C 180,E1 -1952.885,E2 -1952.885} C_VEL
LIN {X 0,Y 714.624,Z 369.984,A -85,B 0,C 180,E1 -1955.837,E2 -1955.837} C_VEL
LIN {X 0,Y 714.076,Z 424.961,A -85,B 0,C 180,E1 -1958.779,E2 -1958.779} C_VEL
LIN {X 0,Y 713.69,Z 470.224,A -85,B 0,C 180,E1 -1961.147,E2 -1961.147} C_VEL
LIN {X 0,Y 714.267,Z 478.095,A -85,B 0,C 180,E1 -1961.253,E2 -1961.253} C_VEL
LIN {X 0,Y 713.764,Z 680.017,A -85,B 0,C 180,E1 -1963.36,E2 -1963.36} C_VEL
LIN {X 0,Y 713.62,Z 699.074,A -85,B 0,C 180,E1 -1963.712,E2 -1963.712} C_VEL
LIN {X 0,Y 713.437,Z 717.391,A -85,B 0,C 180,E1 -1964.201,E2 -1964.201} C_VEL
LIN {X 0,Y 713.216,Z 734.446,A -85,B 0,C 180,E1 -1964.801,E2 -1964.801} C_VEL
LIN {X 0,Y 713.007,Z 751.19,A -85,B 0,C 180,E1 -1965.545,E2 -1965.545} C_VEL
LIN {X 0,Y 712.784,Z 767.054,A -85,B 0,C 180,E1 -1966.41,E2 -1966.41} C_VEL
LIN {X 0,Y 712.567,Z 781.997,A -85,B 0,C 180,E1 -1967.397,E2 -1967.397} C_VEL
LIN {X 0,Y 712.373,Z 795.932,A -85,B 0,C 180,E1 -1968.503,E2 -1968.503} C_VEL
LIN {X 0,Y 712.209,Z 808.757,A -85,B 0,C 180,E1 -1969.729,E2 -1969.729} C_VEL
LIN {X 0,Y 712.087,Z 820.011,A -85,B 0,C 180,E1 -1971.033,E2 -1971.033} C_VEL
LIN {X 0,Y 712.002,Z 829.721,A -85,B 0,C 180,E1 -1972.414,E2 -1972.414} C_VEL
LIN {X 0,Y 711.952,Z 837.452,A -85,B 0,C 180,E1 -1973.792,E2 -1973.792} C_VEL
LIN {X 0,Y 711.927,Z 843.746,A -85,B 0,C 180,E1 -1975.247,E2 -1975.247} C_VEL
LIN {X 0,Y 711.914,Z 848.468,A -85,B 0,C 180,E1 -1976.779,E2 -1976.779} C_VEL
LIN {X 0,Y 711.913,Z 851.342,A -85,B 0,C 180,E1 -1978.31,E2 -1978.31} C_VEL
LIN {X 0,Y 711.913,Z 852.449,A -85,B 0,C 180,E1 -1979.839,E2 -1979.839} C_VEL
LIN {X 0,Y 711.912,Z 851.818,A -85,B 0,C 180,E1 -1981.368,E2 -1981.368} C_VEL
LIN {X 0,Y 711.915,Z 849.433,A -85,B 0,C 180,E1 -1982.898,E2 -1982.898} C_VEL
LIN {X 0,Y 711.923,Z 845.485,A -85,B 0,C 180,E1 -1984.35,E2 -1984.35} C_VEL
LIN {X 0,Y 711.94,Z 839.812,A -85,B 0,C 180,E1 -1985.804,E2 -1985.804} C_VEL
LIN {X 0,Y 711.987,Z 832.719,A -85,B 0,C 180,E1 -1987.18,E2 -1987.18} C_VEL
LIN {X 0,Y 712.053,Z 823.755,A -85,B 0,C 180,E1 -1988.56,E2 -1988.56} C_VEL
LIN {X 0,Y 712.161,Z 813.333,A -85,B 0,C 180,E1 -1989.863,E2 -1989.863} C_VEL
LIN {X 0,Y 712.307,Z 801.092,A -85,B 0,C 180,E1 -1991.124,E2 -1991.124} C_VEL
LIN {X 0,Y 712.491,Z 787.609,A -85,B 0,C 180,E1 -1992.275,E2 -1992.275} C_VEL
LIN {X 0,Y 712.703,Z 772.501,A -85,B 0,C 180,E1 -1993.343,E2 -1993.343} C_VEL
LIN {X 0,Y 712.932,Z 756.541,A -85,B 0,C 180,E1 -1994.273,E2 -1994.273} C_VEL
LIN {X 0,Y 713.137,Z 739.631,A -85,B 0,C 180,E1 -1995.075,E2 -1995.075} C_VEL
LIN {X 0,Y 713.28,Z 729.152,A -85,B 0,C 180,E1 -1995.489,E2 -1995.489} C_VEL
LIN {X 0,Y 712.665,Z 723.159,A -85,B 0,C 180,E1 -1995.719,E2 -1995.719} C_VEL
LIN {X 0,Y 707.093,Z 705.636,A -85,B 0,C 180,E1 -1996.379,E2 -1996.379} C_VEL
LIN {X 0,Y 705.967,Z 698.377,A -85,B 0,C 180,E1 -1996.579,E2 -1996.579} C_VEL
LIN {X 0,Y 705.952,Z 697.308,A -85,B 0,C 180,E1 -1996.603,E2 -1996.603} C_VEL
LIN {X 0,Y 706.113,Z 677.939,A -85,B 0,C 180,E1 -1996.946,E2 -1996.946} C_VEL
LIN {X 0,Y 706.629,Z 474.731,A -85,B 0,C 180,E1 -1999.105,E2 -1999.105} C_VEL
LIN {X 0,Y 705.964,Z 468.931,A -85,B 0,C 180,E1 -1999.205,E2 -1999.205} C_VEL
LIN {X 0,Y 706.627,Z 415.892,A -85,B 0,C 180,E1 -2002.053,E2 -2002.053} C_VEL
LIN {X 0,Y 707.369,Z 358.655,A -85,B 0,C 180,E1 -2005.181,E2 -2005.181} C_VEL
LIN {X 0,Y 708.094,Z 310.205,A -85,B 0,C 180,E1 -2007.875,E2 -2007.875} C_VEL
LIN {X 0,Y 708.987,Z 256.994,A -85,B 0,C 180,E1 -2010.888,E2 -2010.888} C_VEL
LIN {X 0,Y 709.718,Z 212.196,A -85,B 0,C 180,E1 -2013.484,E2 -2013.484} C_VEL
LIN {X 0,Y 704.332,Z 197.5,A -85,B 0,C 180,E1 -2014.65,E2 -2014.65} C_VEL
LIN {X 0,Y 704.344,Z 197.496,A -85,B 0,C 180,E1 -2017.621,E2 -2017.621} C_VEL
LIN {X 0,Y 704.266,Z 197.502,A -85,B 0,C 180,E1 -2020.454,E2 -2020.454} C_VEL
LIN {X 0,Y 704.345,Z 197.496,A -85,B 0,C 180,E1 -2023.289,E2 -2023.289} C_VEL
LIN {X 0,Y 704.333,Z 197.499,A -85,B 0,C 180,E1 -2026.269,E2 -2026.269} C_VEL
LIN {X 0,Y 704.305,Z 197.495,A -85,B 0,C 180,E1 -2029.174,E2 -2029.174} C_VEL
LIN {X 0,Y 704.268,Z 197.504,A -85,B 0,C 180,E1 -2032.272,E2 -2032.272} C_VEL
LIN {X 0,Y 704.339,Z 197.652,A -85,B 0,C 180,E1 -2034.818,E2 -2034.818} C_VEL
LIN {X 0,Y 709.779,Z 213.038,A -85,B 0,C 180,E1 -2036.218,E2 -2036.218} C_VEL
LIN {X 0,Y 708.933,Z 248.718,A -85,B 0,C 180,E1 -2038.78,E2 -2038.78} C_VEL
LIN {X 0,Y 708.094,Z 278.852,A -85,B 0,C 180,E1 -2040.938,E2 -2040.938} C_VEL
LIN {X 0,Y 707.707,Z 304.681,A -85,B 0,C 180,E1 -2042.693,E2 -2042.693} C_VEL
LIN {X 0,Y 709.572,Z 314.84,A -85,B 0,C 180,E1 -2042.884,E2 -2042.884} C_VEL
LIN {X 0,Y 708.323,Z 604.176,A -85,B 0,C 180,E1 -2046.037,E2 -2046.037} C_VEL
LIN {X 0,Y 708.111,Z 623.549,A -85,B 0,C 180,E1 -2046.344,E2 -2046.344} C_VEL
LIN {X 0,Y 707.825,Z 644.177,A -85,B 0,C 180,E1 -2046.802,E2 -2046.802} C_VEL
LIN {X 0,Y 707.416,Z 667.036,A -85,B 0,C 180,E1 -2047.478,E2 -2047.478} C_VEL
LIN {X 0,Y 707.008,Z 686.572,A -85,B 0,C 180,E1 -2048.208,E2 -2048.208} C_VEL
LIN {X 0,Y 706.609,Z 704.141,A -85,B 0,C 180,E1 -2048.992,E2 -2048.992} C_VEL
LIN {X 0,Y 706.199,Z 722.741,A -85,B 0,C 180,E1 -2049.962,E2 -2049.962} C_VEL
LIN {X 0,Y 705.716,Z 742.117,A -85,B 0,C 180,E1 -2051.166,E2 -2051.166} C_VEL
LIN {X 0,Y 705.32,Z 758.277,A -85,B 0,C 180,E1 -2052.339,E2 -2052.339} C_VEL
LIN {X 0,Y 704.961,Z 774.409,A -85,B 0,C 180,E1 -2053.69,E2 -2053.69} C_VEL
LIN {X 0,Y 704.623,Z 790.595,A -85,B 0,C 180,E1 -2055.285,E2 -2055.285} C_VEL
LIN {X 0,Y 704.384,Z 802.926,A -85,B 0,C 180,E1 -2056.705,E2 -2056.705} C_VEL
LIN {X 0,Y 704.202,Z 814.074,A -85,B 0,C 180,E1 -2058.202,E2 -2058.202} C_VEL
LIN {X 0,Y 704.077,Z 824.984,A -85,B 0,C 180,E1 -2059.94,E2 -2059.94} C_VEL
LIN {X 0,Y 703.991,Z 833.448,A -85,B 0,C 180,E1 -2061.588,E2 -2061.588} C_VEL
LIN {X 0,Y 703.935,Z 839.935,A -85,B 0,C 180,E1 -2063.162,E2 -2063.162} C_VEL
LIN {X 0,Y 703.916,Z 845.471,A -85,B 0,C 180,E1 -2064.866,E2 -2064.866} C_VEL
LIN {X 0,Y 703.903,Z 849.66,A -85,B 0,C 180,E1 -2066.743,E2 -2066.743} C_VEL
LIN {X 0,Y 703.9,Z 851.844,A -85,B 0,C 180,E1 -2068.535,E2 -2068.535} C_VEL
LIN {X 0,Y 703.902,Z 852.452,A -85,B 0,C 180,E1 -2070.326,E2 -2070.326} C_VEL
LIN {X 0,Y 703.911,Z 851.29,A -85,B 0,C 180,E1 -2072.198,E2 -2072.198} C_VEL
LIN {X 0,Y 703.919,Z 848.414,A -85,B 0,C 180,E1 -2073.991,E2 -2073.991} C_VEL
LIN {X 0,Y 703.925,Z 843.802,A -85,B 0,C 180,E1 -2075.788,E2 -2075.788} C_VEL
LIN {X 0,Y 703.954,Z 837.441,A -85,B 0,C 180,E1 -2077.591,E2 -2077.591} C_VEL
LIN {X 0,Y 704.021,Z 829.494,A -85,B 0,C 180,E1 -2079.318,E2 -2079.318} C_VEL
LIN {X 0,Y 704.122,Z 820.083,A -85,B 0,C 180,E1 -2080.969,E2 -2080.969} C_VEL
LIN {X 0,Y 704.287,Z 809.445,A -85,B 0,C 180,E1 -2082.546,E2 -2082.546} C_VEL
LIN {X 0,Y 704.516,Z 795.925,A -85,B 0,C 180,E1 -2084.22,E2 -2084.22} C_VEL
LIN {X 0,Y 704.779,Z 782.443,A -85,B 0,C 180,E1 -2085.638,E2 -2085.638} C_VEL
LIN {X 0,Y 705.124,Z 767.259,A -85,B 0,C 180,E1 -2087.027,E2 -2087.027} C_VEL
LIN {X 0,Y 705.535,Z 749.3,A -85,B 0,C 180,E1 -2088.423,E2 -2088.423} C_VEL
LIN {X 0,Y 705.94,Z 732.752,A -85,B 0,C 180,E1 -2089.528,E2 -2089.528} C_VEL
LIN {X 0,Y 706.371,Z 714.967,A -85,B 0,C 180,E1 -2090.552,E2 -2090.552} C_VEL
LIN {X 0,Y 706.858,Z 693.799,A -85,B 0,C 180,E1 -2091.579,E2 -2091.579} C_VEL
LIN {X 0,Y 707.285,Z 673.767,A -85,B 0,C 180,E1 -2092.376,E2 -2092.376} C_VEL
LIN {X 0,Y 707.599,Z 655.35,A -85,B 0,C 180,E1 -2092.977,E2 -2092.977} C_VEL
LIN {X 0,Y 707.945,Z 636.235,A -85,B 0,C 180,E1 -2093.48,E2 -2093.48} C_VEL
LIN {X 0,Y 708.226,Z 614.339,A -85,B 0,C 180,E1 -2093.912,E2 -2093.912} C_VEL
LIN {X 0,Y 708.439,Z 584.242,A -85,B 0,C 180,E1 -2094.283,E2 -2094.283} C_VEL
LIN {X 0,Y 709.568,Z 313.73,A -85,B 0,C 180,E1 -2097.218,E2 -2097.218} C_VEL
LIN {X 0,Y 707.643,Z 303.896,A -85,B 0,C 180,E1 -2097.428,E2 -2097.428} C_VEL
LIN {X 0,Y 708.447,Z 263.895,A -85,B 0,C 180,E1 -2100.209,E2 -2100.209} C_VEL
LIN {X 0,Y 709.423,Z 230.579,A -85,B 0,C 180,E1 -2102.623,E2 -2102.623} C_VEL
LIN {X 0,Y 709.669,Z 212.635,A -85,B 0,C 180,E1 -2103.914,E2 -2103.914} C_VEL
LIN {X 0,Y 704.312,Z 197.503,A -85,B 0,C 180,E1 -2105.296,E2 -2105.296} C_VEL
LIN {X 0,Y 704.342,Z 197.493,A -85,B 0,C 180,E1 -2108.343,E2 -2108.343} C_VEL
LIN {X 0,Y 704.315,Z 197.496,A -85,B 0,C 180,E1 -2111.322,E2 -2111.322} C_VEL
LIN {X 0,Y 704.337,Z 197.493,A -85,B 0,C 180,E1 -2114.316,E2 -2114.316} C_VEL
LIN {X 0,Y 704.312,Z 197.494,A -85,B 0,C 180,E1 -2117.265,E2 -2117.265} C_VEL
LIN {X 0,Y 704.329,Z 197.494,A -85,B 0,C 180,E1 -2120.177,E2 -2120.177} C_VEL
LIN {X 0,Y 704.314,Z 197.491,A -85,B 0,C 180,E1 -2123.093,E2 -2123.093} C_VEL
LIN {X 0,Y 704.33,Z 197.492,A -85,B 0,C 180,E1 -2126.003,E2 -2126.003} C_VEL
LIN {X 0,Y 704.321,Z 197.491,A -85,B 0,C 180,E1 -2128.98,E2 -2128.98} C_VEL
LIN {X 0,Y 704.336,Z 197.494,A -85,B 0,C 180,E1 -2131.88,E2 -2131.88} C_VEL
LIN {X 0,Y 704.331,Z 197.488,A -85,B 0,C 180,E1 -2134.921,E2 -2134.921} C_VEL
LIN {X 0,Y 704.335,Z 197.498,A -85,B 0,C 180,E1 -2137.901,E2 -2137.901} C_VEL
LIN {X 0,Y 704.334,Z 197.485,A -85,B 0,C 180,E1 -2140.943,E2 -2140.943} C_VEL
LIN {X 0,Y 704.331,Z 197.497,A -85,B 0,C 180,E1 -2143.964,E2 -2143.964} C_VEL
LIN {X 0,Y 704.339,Z 197.483,A -85,B 0,C 180,E1 -2146.955,E2 -2146.955} C_VEL
LIN {X 0,Y 704.326,Z 197.497,A -85,B 0,C 180,E1 -2150.026,E2 -2150.026} C_VEL
LIN {X 0,Y 704.34,Z 197.484,A -85,B 0,C 180,E1 -2152.987,E2 -2152.987} C_VEL
LIN {X 0,Y 704.327,Z 197.498,A -85,B 0,C 180,E1 -2156.011,E2 -2156.011} C_VEL
LIN {X 0,Y 704.342,Z 197.486,A -85,B 0,C 180,E1 -2159.024,E2 -2159.024} C_VEL
LIN {X 0,Y 704.326,Z 197.497,A -85,B 0,C 180,E1 -2162.034,E2 -2162.034} C_VEL
LIN {X 0,Y 704.338,Z 197.488,A -85,B 0,C 180,E1 -2165.05,E2 -2165.05} C_VEL
LIN {X 0,Y 704.322,Z 197.495,A -85,B 0,C 180,E1 -2168.079,E2 -2168.079} C_VEL
LIN {X 0,Y 704.335,Z 197.489,A -85,B 0,C 180,E1 -2171.049,E2 -2171.049} C_VEL
LIN {X 0,Y 704.317,Z 197.497,A -85,B 0,C 180,E1 -2174.157,E2 -2174.157} C_VEL
LIN {X 0,Y 704.333,Z 197.49,A -85,B 0,C 180,E1 -2177.089,E2 -2177.089} C_VEL
LIN {X 0,Y 704.315,Z 197.497,A -85,B 0,C 180,E1 -2180.181,E2 -2180.181} C_VEL
LIN {X 0,Y 704.324,Z 197.491,A -85,B 0,C 180,E1 -2183.084,E2 -2183.084} C_VEL
LIN {X 0,Y 704.313,Z 197.496,A -85,B 0,C 180,E1 -2186.204,E2 -2186.204} C_VEL
LIN {X 0,Y 704.314,Z 197.491,A -85,B 0,C 180,E1 -2189.047,E2 -2189.047} C_VEL
LIN {X 0,Y 704.311,Z 197.499,A -85,B 0,C 180,E1 -2192.207,E2 -2192.207} C_VEL
LIN {X 0,Y 704.301,Z 197.494,A -85,B 0,C 180,E1 -2194.999,E2 -2194.999} C_VEL
LIN {X 0,Y 704.332,Z 197.497,A -85,B 0,C 180,E1 -2198.034,E2 -2198.034} C_VEL
LIN {X 0,Y 704.286,Z 197.496,A -85,B 0,C 180,E1 -2200.825,E2 -2200.825} C_VEL
LIN {X 0,Y 704.345,Z 197.495,A -85,B 0,C 180,E1 -2203.737,E2 -2203.737} C_VEL
LIN {X 0,Y 704.283,Z 197.501,A -85,B 0,C 180,E1 -2206.628,E2 -2206.628} C_VEL
LIN {X 0,Y 704.318,Z 197.608,A -85,B 0,C 180,E1 -2209.236,E2 -2209.236} C_VEL
LIN {X 0,Y 705.292,Z 200.424,A -85,B 0,C 180,E1 -2209.454,E2 -2209.454} C_VEL
LIN {X 0,Y 706.704,Z 203.245,A -85,B 0,C 180,E1 -2209.695,E2 -2209.695} C_VEL
LIN {X 0,Y 713.285,Z 217.385,A -85,B 0,C 180,E1 -2210.824,E2 -2210.824} C_VEL
LIN {X 0,Y 712.298,Z 270.275,A -85,B 0,C 180,E1 -2213.318,E2 -2213.318} C_VEL
LIN {X 0,Y 711.848,Z 299.334,A -85,B 0,C 180,E1 -2214.644,E2 -2214.644} C_VEL
LIN {X 0,Y 713.279,Z 309.701,A -85,B 0,C 180,E1 -2214.85,E2 -2214.85} C_VEL
LIN {X 0,Y 711.768,Z 574.626,A -85,B 0,C 180,E1 -2217.911,E2 -2217.911} C_VEL
LIN {X 0,Y 711.095,Z 691.218,A -85,B 0,C 180,E1 -2219.254,E2 -2219.254} C_VEL
LIN {X 0,Y 710.694,Z 716.763,A -85,B 0,C 180,E1 -2219.695,E2 -2219.695} C_VEL
LIN {X 0,Y 710.27,Z 738.453,A -85,B 0,C 180,E1 -2220.205,E2 -2220.205} C_VEL
LIN {X 0,Y 709.758,Z 762.564,A -85,B 0,C 180,E1 -2220.92,E2 -2220.92} C_VEL
LIN {X 0,Y 709.159,Z 784.49,A -85,B 0,C 180,E1 -2221.722,E2 -2221.722} C_VEL
LIN {X 0,Y 708.561,Z 807.17,A -85,B 0,C 180,E1 -2222.702,E2 -2222.702} C_VEL
LIN {X 0,Y 707.877,Z 828.76,A -85,B 0,C 180,E1 -2223.806,E2 -2223.806} C_VEL
LIN {X 0,Y 707.237,Z 849.752,A -85,B 0,C 180,E1 -2225.038,E2 -2225.038} C_VEL
LIN {X 0,Y 706.624,Z 869.053,A -85,B 0,C 180,E1 -2226.349,E2 -2226.349} C_VEL
LIN {X 0,Y 706.064,Z 887.763,A -85,B 0,C 180,E1 -2227.783,E2 -2227.783} C_VEL
LIN {X 0,Y 705.564,Z 904.786,A -85,B 0,C 180,E1 -2229.281,E2 -2229.281} C_VEL
LIN {X 0,Y 705.127,Z 920.967,A -85,B 0,C 180,E1 -2230.879,E2 -2230.879} C_VEL
LIN {X 0,Y 704.764,Z 935.224,A -85,B 0,C 180,E1 -2232.496,E2 -2232.496} C_VEL
LIN {X 0,Y 704.49,Z 949.061,A -85,B 0,C 180,E1 -2234.271,E2 -2234.271} C_VEL
LIN {X 0,Y 704.274,Z 960.798,A -85,B 0,C 180,E1 -2236.033,E2 -2236.033} C_VEL
LIN {X 0,Y 704.126,Z 971.406,A -85,B 0,C 180,E1 -2237.868,E2 -2237.868} C_VEL
LIN {X 0,Y 704.018,Z 980.722,A -85,B 0,C 180,E1 -2239.817,E2 -2239.817} C_VEL
LIN {X 0,Y 703.942,Z 987.424,A -85,B 0,C 180,E1 -2241.505,E2 -2241.505} C_VEL
LIN {X 0,Y 703.916,Z 993.864,A -85,B 0,C 180,E1 -2243.557,E2 -2243.557} C_VEL
LIN {X 0,Y 703.915,Z 997.973,A -85,B 0,C 180,E1 -2245.356,E2 -2245.356} C_VEL
LIN {X 0,Y 703.884,Z 1000.91,A -85,B 0,C 180,E1 -2247.232,E2 -2247.232} C_VEL
LIN {X 0,Y 703.888,Z 1002.284,A -85,B 0,C 180,E1 -2249.186,E2 -2249.186} C_VEL
LIN {X 0,Y 703.888,Z 1002.284,A -85,B 0,C 180,E1 -2250.814,E2 -2250.814} C_VEL
LIN {X 0,Y 703.884,Z 1000.909,A -85,B 0,C 180,E1 -2252.768,E2 -2252.768} C_VEL
LIN {X 0,Y 703.916,Z 997.972,A -85,B 0,C 180,E1 -2254.644,E2 -2254.644} C_VEL
LIN {X 0,Y 703.917,Z 993.864,A -85,B 0,C 180,E1 -2256.443,E2 -2256.443} C_VEL
LIN {X 0,Y 703.94,Z 987.423,A -85,B 0,C 180,E1 -2258.495,E2 -2258.495} C_VEL
LIN {X 0,Y 704.019,Z 980.721,A -85,B 0,C 180,E1 -2260.184,E2 -2260.184} C_VEL
LIN {X 0,Y 704.126,Z 971.406,A -85,B 0,C 180,E1 -2262.132,E2 -2262.132} C_VEL
LIN {X 0,Y 704.275,Z 960.8,A -85,B 0,C 180,E1 -2263.967,E2 -2263.967} C_VEL
LIN {X 0,Y 704.504,Z 948.438,A -85,B 0,C 180,E1 -2265.813,E2 -2265.813} C_VEL
LIN {X 0,Y 704.764,Z 935.223,A -85,B 0,C 180,E1 -2267.504,E2 -2267.504} C_VEL
LIN {X 0,Y 705.146,Z 920.174,A -85,B 0,C 180,E1 -2269.207,E2 -2269.207} C_VEL
LIN {X 0,Y 705.602,Z 903.533,A -85,B 0,C 180,E1 -2270.836,E2 -2270.836} C_VEL
LIN {X 0,Y 706.116,Z 885.605,A -85,B 0,C 180,E1 -2272.39,E2 -2272.39} C_VEL
LIN {X 0,Y 706.66,Z 868.004,A -85,B 0,C 180,E1 -2273.726,E2 -2273.726} C_VEL
LIN {X 0,Y 707.288,Z 847.62,A -85,B 0,C 180,E1 -2275.094,E2 -2275.094} C_VEL
LIN {X 0,Y 707.909,Z 827.83,A -85,B 0,C 180,E1 -2276.245,E2 -2276.245} C_VEL
LIN {X 0,Y 708.585,Z 806.236,A -85,B 0,C 180,E1 -2277.343,E2 -2277.343} C_VEL
LIN {X 0,Y 709.159,Z 784.489,A -85,B 0,C 180,E1 -2278.278,E2 -2278.278} C_VEL
LIN {X 0,Y 709.757,Z 762.561,A -85,B 0,C 180,E1 -2279.08,E2 -2279.08} C_VEL
LIN {X 0,Y 710.273,Z 738.223,A -85,B 0,C 180,E1 -2279.801,E2 -2279.801} C_VEL
LIN {X 0,Y 710.707,Z 716.369,A -85,B 0,C 180,E1 -2280.313,E2 -2280.313} C_VEL
LIN {X 0,Y 711.096,Z 691.06,A -85,B 0,C 180,E1 -2280.748,E2 -2280.748} C_VEL
LIN {X 0,Y 711.957,Z 541.029,A -85,B 0,C 180,E1 -2282.472,E2 -2282.472} C_VEL
LIN {X 0,Y 713.246,Z 308.067,A -85,B 0,C 180,E1 -2285.171,E2 -2285.171} C_VEL
LIN {X 0,Y 711.737,Z 298.171,A -85,B 0,C 180,E1 -2285.391,E2 -2285.391} C_VEL
LIN {X 0,Y 712.953,Z 237.759,A -85,B 0,C 180,E1 -2288.206,E2 -2288.206} C_VEL
LIN {X 0,Y 713.036,Z 216.483,A -85,B 0,C 180,E1 -2289.215,E2 -2289.215} C_VEL
LIN {X 0,Y 705.587,Z 200.909,A -85,B 0,C 180,E1 -2290.576,E2 -2290.576} C_VEL
LIN {X 0,Y 704.305,Z 197.503,A -85,B 0,C 180,E1 -2290.88,E2 -2290.88} C_VEL
LIN {X 0,Y 704.31,Z 197.502,A -85,B 0,C 180,E1 -2293.627,E2 -2293.627} C_VEL
LIN {X 0,Y 704.336,Z 197.497,A -85,B 0,C 180,E1 -2296.623,E2 -2296.623} C_VEL
LIN {X 0,Y 704.295,Z 197.503,A -85,B 0,C 180,E1 -2299.549,E2 -2299.549} C_VEL
LIN {X 0,Y 704.343,Z 197.497,A -85,B 0,C 180,E1 -2302.52,E2 -2302.52} C_VEL
LIN {X 0,Y 704.326,Z 197.661,A -85,B 0,C 180,E1 -2305.159,E2 -2305.159} C_VEL
LIN {X 0,Y 705.506,Z 200.851,A -85,B 0,C 180,E1 -2305.465,E2 -2305.465} C_VEL
LIN {X 0,Y 710.491,Z 213.304,A -85,B 0,C 180,E1 -2306.615,E2 -2306.615} C_VEL
LIN {X 0,Y 708.907,Z 262.138,A -85,B 0,C 180,E1 -2309.519,E2 -2309.519} C_VEL
LIN {X 0,Y 707.787,Z 319.047,A -85,B 0,C 180,E1 -2312.76,E2 -2312.76} C_VEL
LIN {X 0,Y 707.075,Z 372.246,A -85,B 0,C 180,E1 -2315.7,E2 -2315.7} C_VEL
LIN {X 0,Y 706.42,Z 427.117,A -85,B 0,C 180,E1 -2318.668,E2 -2318.668} C_VEL
LIN {X 0,Y 706.013,Z 467.654,A -85,B 0,C 180,E1 -2320.807,E2 -2320.807} C_VEL
LIN {X 0,Y 707.031,Z 478.159,A -85,B 0,C 180,E1 -2320.977,E2 -2320.977} C_VEL
LIN {X 0,Y 706.228,Z 638.86,A -85,B 0,C 180,E1 -2322.716,E2 -2322.716} C_VEL
LIN {X 0,Y 706.078,Z 681.387,A -85,B 0,C 180,E1 -2323.195,E2 -2323.195} C_VEL
LIN {X 0,Y 705.91,Z 700.233,A -85,B 0,C 180,E1 -2323.556,E2 -2323.556} C_VEL
LIN {X 0,Y 705.703,Z 718.075,A -85,B 0,C 180,E1 -2324.045,E2 -2324.045} C_VEL
LIN {X 0,Y 705.433,Z 735.675,A -85,B 0,C 180,E1 -2324.681,E2 -2324.681} C_VEL
LIN {X 0,Y 705.18,Z 752.818,A -85,B 0,C 180,E1 -2325.465,E2 -2325.465} C_VEL
LIN {X 0,Y 704.907,Z 769.061,A -85,B 0,C 180,E1 -2326.381,E2 -2326.381} C_VEL
LIN {X 0,Y 704.65,Z 784.222,A -85,B 0,C 180,E1 -2327.419,E2 -2327.419} C_VEL
LIN {X 0,Y 704.43,Z 797.789,A -85,B 0,C 180,E1 -2328.538,E2 -2328.538} C_VEL
LIN {X 0,Y 704.246,Z 810.301,A -85,B 0,C 180,E1 -2329.777,E2 -2329.777} C_VEL
LIN {X 0,Y 704.107,Z 821.284,A -85,B 0,C 180,E1 -2331.095,E2 -2331.095} C_VEL
LIN {X 0,Y 704.013,Z 830.753,A -85,B 0,C 180,E1 -2332.492,E2 -2332.492} C_VEL
LIN {X 0,Y 703.96,Z 838.264,A -85,B 0,C 180,E1 -2333.885,E2 -2333.885} C_VEL
LIN {X 0,Y 703.926,Z 844.352,A -85,B 0,C 180,E1 -2335.356,E2 -2335.356} C_VEL
LIN {X 0,Y 703.915,Z 848.674,A -85,B 0,C 180,E1 -2336.824,E2 -2336.824} C_VEL
LIN {X 0,Y 703.911,Z 851.455,A -85,B 0,C 180,E1 -2338.372,E2 -2338.372} C_VEL
LIN {X 0,Y 703.916,Z 852.472,A -85,B 0,C 180,E1 -2339.919,E2 -2339.919} C_VEL
LIN {X 0,Y 703.909,Z 851.748,A -85,B 0,C 180,E1 -2341.465,E2 -2341.465} C_VEL
LIN {X 0,Y 703.92,Z 849.201,A -85,B 0,C 180,E1 -2343.048,E2 -2343.048} C_VEL
LIN {X 0,Y 703.924,Z 844.972,A -85,B 0,C 180,E1 -2344.562,E2 -2344.562} C_VEL
LIN {X 0,Y 703.954,Z 839.101,A -85,B 0,C 180,E1 -2346.033,E2 -2346.033} C_VEL
LIN {X 0,Y 704.011,Z 831.315,A -85,B 0,C 180,E1 -2347.508,E2 -2347.508} C_VEL
LIN {X 0,Y 704.104,Z 821.977,A -85,B 0,C 180,E1 -2348.905,E2 -2348.905} C_VEL
LIN {X 0,Y 704.234,Z 811.14,A -85,B 0,C 180,E1 -2350.223,E2 -2350.223} C_VEL
LIN {X 0,Y 704.415,Z 798.793,A -85,B 0,C 180,E1 -2351.462,E2 -2351.462} C_VEL
LIN {X 0,Y 704.628,Z 785.421,A -85,B 0,C 180,E1 -2352.581,E2 -2352.581} C_VEL
LIN {X 0,Y 704.88,Z 770.501,A -85,B 0,C 180,E1 -2353.62,E2 -2353.62} C_VEL
LIN {X 0,Y 705.151,Z 754.561,A -85,B 0,C 180,E1 -2354.536,E2 -2354.536} C_VEL
LIN {X 0,Y 705.4,Z 737.341,A -85,B 0,C 180,E1 -2355.34,E2 -2355.34} C_VEL
LIN {X 0,Y 705.688,Z 719.079,A -85,B 0,C 180,E1 -2356.012,E2 -2356.012} C_VEL
LIN {X 0,Y 705.901,Z 700.559,A -85,B 0,C 180,E1 -2356.526,E2 -2356.526} C_VEL
LIN {X 0,Y 705.952,Z 697.308,A -85,B 0,C 180,E1 -2356.603,E2 -2356.603} C_VEL
LIN {X 0,Y 705.12,Z 689.881,A -85,B 0,C 180,E1 -2356.776,E2 -2356.776} C_VEL
LIN {X 0,Y 699.513,Z 671.284,A -85,B 0,C 180,E1 -2357.201,E2 -2357.201} C_VEL
LIN {X 0,Y 698.559,Z 663.716,A -85,B 0,C 180,E1 -2357.312,E2 -2357.312} C_VEL
LIN {X 0,Y 699.205,Z 475.631,A -85,B 0,C 180,E1 -2359.339,E2 -2359.339} C_VEL
LIN {X 0,Y 698.318,Z 468.147,A -85,B 0,C 180,E1 -2359.467,E2 -2359.467} C_VEL
LIN {X 0,Y 699.133,Z 412.338,A -85,B 0,C 180,E1 -2362.497,E2 -2362.497} C_VEL
LIN {X 0,Y 699.946,Z 357.952,A -85,B 0,C 180,E1 -2365.505,E2 -2365.505} C_VEL
LIN {X 0,Y 700.769,Z 309.425,A -85,B 0,C 180,E1 -2368.229,E2 -2368.229} C_VEL
LIN {X 0,Y 701.828,Z 255.192,A -85,B 0,C 180,E1 -2371.333,E2 -2371.333} C_VEL
LIN {X 0,Y 702.54,Z 215.212,A -85,B 0,C 180,E1 -2373.673,E2 -2373.673} C_VEL
LIN {X 0,Y 696.388,Z 198.488,A -85,B 0,C 180,E1 -2375.025,E2 -2375.025} C_VEL
LIN {X 0,Y 696.382,Z 198.488,A -85,B 0,C 180,E1 -2378.023,E2 -2378.023} C_VEL
LIN {X 0,Y 696.341,Z 198.491,A -85,B 0,C 180,E1 -2380.794,E2 -2380.794} C_VEL
LIN {X 0,Y 696.374,Z 198.485,A -85,B 0,C 180,E1 -2383.879,E2 -2383.879} C_VEL
LIN {X 0,Y 696.382,Z 198.485,A -85,B 0,C 180,E1 -2386.773,E2 -2386.773} C_VEL
LIN {X 0,Y 696.407,Z 198.487,A -85,B 0,C 180,E1 -2389.804,E2 -2389.804} C_VEL
LIN {X 0,Y 696.335,Z 198.493,A -85,B 0,C 180,E1 -2392.704,E2 -2392.704} C_VEL
LIN {X 0,Y 696.386,Z 198.717,A -85,B 0,C 180,E1 -2394.397,E2 -2394.397} C_VEL
LIN {X 0,Y 702.777,Z 216.31,A -85,B 0,C 180,E1 -2396.03,E2 -2396.03} C_VEL
LIN {X 0,Y 701.834,Z 254.954,A -85,B 0,C 180,E1 -2398.81,E2 -2398.81} C_VEL
LIN {X 0,Y 700.991,Z 278.35,A -85,B 0,C 180,E1 -2400.521,E2 -2400.521} C_VEL
LIN {X 0,Y 700.376,Z 296.666,A -85,B 0,C 180,E1 -2401.846,E2 -2401.846} C_VEL
LIN {X 0,Y 700.324,Z 304.737,A -85,B 0,C 180,E1 -2402.381,E2 -2402.381} C_VEL
LIN {X 0,Y 702.442,Z 316.284,A -85,B 0,C 180,E1 -2402.602,E2 -2402.602} C_VEL
LIN {X 0,Y 701.01,Z 603.766,A -85,B 0,C 180,E1 -2405.765,E2 -2405.765} C_VEL
LIN {X 0,Y 700.785,Z 622.516,A -85,B 0,C 180,E1 -2406.062,E2 -2406.062} C_VEL
LIN {X 0,Y 700.461,Z 642.006,A -85,B 0,C 180,E1 -2406.488,E2 -2406.488} C_VEL
LIN {X 0,Y 700.045,Z 664.513,A -85,B 0,C 180,E1 -2407.138,E2 -2407.138} C_VEL
LIN {X 0,Y 699.549,Z 684.387,A -85,B 0,C 180,E1 -2407.87,E2 -2407.87} C_VEL
LIN {X 0,Y 699.109,Z 702.07,A -85,B 0,C 180,E1 -2408.654,E2 -2408.654} C_VEL
LIN {X 0,Y 698.667,Z 718.036,A -85,B 0,C 180,E1 -2409.474,E2 -2409.474} C_VEL
LIN {X 0,Y 698.192,Z 736.124,A -85,B 0,C 180,E1 -2410.551,E2 -2410.551} C_VEL
LIN {X 0,Y 697.638,Z 755.555,A -85,B 0,C 180,E1 -2411.923,E2 -2411.923} C_VEL
LIN {X 0,Y 697.214,Z 771.068,A -85,B 0,C 180,E1 -2413.203,E2 -2413.203} C_VEL
LIN {X 0,Y 696.867,Z 784.942,A -85,B 0,C 180,E1 -2414.521,E2 -2414.521} C_VEL
LIN {X 0,Y 696.552,Z 799.52,A -85,B 0,C 180,E1 -2416.13,E2 -2416.13} C_VEL
LIN {X 0,Y 696.312,Z 811.743,A -85,B 0,C 180,E1 -2417.73,E2 -2417.73} C_VEL
LIN {X 0,Y 696.144,Z 821.645,A -85,B 0,C 180,E1 -2419.251,E2 -2419.251} C_VEL
LIN {X 0,Y 696.03,Z 831.1,A -85,B 0,C 180,E1 -2420.991,E2 -2420.991} C_VEL
LIN {X 0,Y 695.962,Z 838.667,A -85,B 0,C 180,E1 -2422.737,E2 -2422.737} C_VEL
LIN {X 0,Y 695.924,Z 844.024,A -85,B 0,C 180,E1 -2424.31,E2 -2424.31} C_VEL
LIN {X 0,Y 695.918,Z 848.562,A -85,B 0,C 180,E1 -2426.128,E2 -2426.128} C_VEL
LIN {X 0,Y 695.917,Z 851.512,A -85,B 0,C 180,E1 -2428.106,E2 -2428.106} C_VEL
LIN {X 0,Y 695.913,Z 852.449,A -85,B 0,C 180,E1 -2429.918,E2 -2429.918} C_VEL
LIN {X 0,Y 695.906,Z 851.784,A -85,B 0,C 180,E1 -2431.647,E2 -2431.647} C_VEL
LIN {X 0,Y 695.907,Z 849.522,A -85,B 0,C 180,E1 -2433.46,E2 -2433.46} C_VEL
LIN {X 0,Y 695.924,Z 845.248,A -85,B 0,C 180,E1 -2435.359,E2 -2435.359} C_VEL
LIN {X 0,Y 695.943,Z 839.908,A -85,B 0,C 180,E1 -2437.015,E2 -2437.015} C_VEL
LIN {X 0,Y 696.003,Z 833.105,A -85,B 0,C 180,E1 -2438.676,E2 -2438.676} C_VEL
LIN {X 0,Y 696.131,Z 823.641,A -85,B 0,C 180,E1 -2440.511,E2 -2440.511} C_VEL
LIN {X 0,Y 696.282,Z 812.959,A -85,B 0,C 180,E1 -2442.187,E2 -2442.187} C_VEL
LIN {X 0,Y 696.493,Z 801.626,A -85,B 0,C 180,E1 -2443.702,E2 -2443.702} C_VEL
LIN {X 0,Y 696.818,Z 787.532,A -85,B 0,C 180,E1 -2445.309,E2 -2445.309} C_VEL
LIN {X 0,Y 697.194,Z 772.08,A -85,B 0,C 180,E1 -2446.797,E2 -2446.797} C_VEL
LIN {X 0,Y 697.605,Z 756.696,A -85,B 0,C 180,E1 -2448.078,E2 -2448.078} C_VEL
LIN {X 0,Y 698.113,Z 738.816,A -85,B 0,C 180,E1 -2449.364,E2 -2449.364} C_VEL
LIN {X 0,Y 698.603,Z 720.712,A -85,B 0,C 180,E1 -2450.468,E2 -2450.468} C_VEL
LIN {X 0,Y 699.059,Z 703.818,A -85,B 0,C 180,E1 -2451.352,E2 -2451.352} C_VEL
LIN {X 0,Y 699.505,Z 686.317,A -85,B 0,C 180,E1 -2452.139,E2 -2452.139} C_VEL
LIN {X 0,Y 699.98,Z 666.792,A -85,B 0,C 180,E1 -2452.874,E2 -2452.874} C_VEL
LIN {X 0,Y 700.453,Z 642.92,A -85,B 0,C 180,E1 -2453.579,E2 -2453.579} C_VEL
LIN {X 0,Y 700.777,Z 623.133,A -85,B 0,C 180,E1 -2454.017,E2 -2454.017} C_VEL
LIN {X 0,Y 701.005,Z 604.319,A -85,B 0,C 180,E1 -2454.318,E2 -2454.318} C_VEL
LIN {X 0,Y 702.395,Z 324.273,A -85,B 0,C 180,E1 -2457.4,E2 -2457.4} C_VEL
LIN {X 0,Y 702.223,Z 314.026,A -85,B 0,C 180,E1 -2457.523,E2 -2457.523} C_VEL
LIN {X 0,Y 700.249,Z 303.888,A -85,B 0,C 180,E1 -2457.742,E2 -2457.742} C_VEL
LIN {X 0,Y 700.856,Z 281.358,A -85,B 0,C 180,E1 -2459.343,E2 -2459.343} C_VEL
LIN {X 0,Y 701.642,Z 260.693,A -85,B 0,C 180,E1 -2460.866,E2 -2460.866} C_VEL
LIN {X 0,Y 702.661,Z 224.057,A -85,B 0,C 180,E1 -2463.513,E2 -2463.513} C_VEL
LIN {X 0,Y 702.674,Z 215.893,A -85,B 0,C 180,E1 -2464.101,E2 -2464.101} C_VEL
LIN {X 0,Y 697.029,Z 200.774,A -85,B 0,C 180,E1 -2465.519,E2 -2465.519} C_VEL
LIN {X 0,Y 696.4,Z 198.489,A -85,B 0,C 180,E1 -2465.731,E2 -2465.731} C_VEL
LIN {X 0,Y 696.376,Z 198.485,A -85,B 0,C 180,E1 -2468.77,E2 -2468.77} C_VEL
LIN {X 0,Y 696.405,Z 198.485,A -85,B 0,C 180,E1 -2471.702,E2 -2471.702} C_VEL
LIN {X 0,Y 696.387,Z 198.482,A -85,B 0,C 180,E1 -2474.713,E2 -2474.713} C_VEL
LIN {X 0,Y 696.402,Z 198.488,A -85,B 0,C 180,E1 -2477.683,E2 -2477.683} C_VEL
LIN {X 0,Y 696.393,Z 198.479,A -85,B 0,C 180,E1 -2480.714,E2 -2480.714} C_VEL
LIN {X 0,Y 696.401,Z 198.484,A -85,B 0,C 180,E1 -2483.796,E2 -2483.796} C_VEL
LIN {X 0,Y 696.39,Z 198.474,A -85,B 0,C 180,E1 -2486.835,E2 -2486.835} C_VEL
LIN {X 0,Y 696.402,Z 198.485,A -85,B 0,C 180,E1 -2489.832,E2 -2489.832} C_VEL
LIN {X 0,Y 696.391,Z 198.476,A -85,B 0,C 180,E1 -2492.899,E2 -2492.899} C_VEL
LIN {X 0,Y 696.393,Z 198.477,A -85,B 0,C 180,E1 -2495.948,E2 -2495.948} C_VEL
LIN {X 0,Y 696.394,Z 198.477,A -85,B 0,C 180,E1 -2498.964,E2 -2498.964} C_VEL
LIN {X 0,Y 696.393,Z 198.478,A -85,B 0,C 180,E1 -2501.932,E2 -2501.932} C_VEL
LIN {X 0,Y 696.401,Z 198.476,A -85,B 0,C 180,E1 -2504.937,E2 -2504.937} C_VEL
LIN {X 0,Y 696.389,Z 198.479,A -85,B 0,C 180,E1 -2507.983,E2 -2507.983} C_VEL
LIN {X 0,Y 696.399,Z 198.477,A -85,B 0,C 180,E1 -2510.996,E2 -2510.996} C_VEL
LIN {X 0,Y 696.39,Z 198.478,A -85,B 0,C 180,E1 -2513.983,E2 -2513.983} C_VEL
LIN {X 0,Y 696.4,Z 198.477,A -85,B 0,C 180,E1 -2517.037,E2 -2517.037} C_VEL
LIN {X 0,Y 696.383,Z 198.475,A -85,B 0,C 180,E1 -2520.082,E2 -2520.082} C_VEL
LIN {X 0,Y 696.399,Z 198.476,A -85,B 0,C 180,E1 -2523.045,E2 -2523.045} C_VEL
LIN {X 0,Y 696.381,Z 198.477,A -85,B 0,C 180,E1 -2526.099,E2 -2526.099} C_VEL
LIN {X 0,Y 696.401,Z 198.475,A -85,B 0,C 180,E1 -2529.087,E2 -2529.087} C_VEL
LIN {X 0,Y 696.376,Z 198.486,A -85,B 0,C 180,E1 -2532.185,E2 -2532.185} C_VEL
LIN {X 0,Y 696.402,Z 198.477,A -85,B 0,C 180,E1 -2535.148,E2 -2535.148} C_VEL
LIN {X 0,Y 696.37,Z 198.485,A -85,B 0,C 180,E1 -2538.241,E2 -2538.241} C_VEL
LIN {X 0,Y 696.401,Z 198.478,A -85,B 0,C 180,E1 -2541.212,E2 -2541.212} C_VEL
LIN {X 0,Y 696.37,Z 198.486,A -85,B 0,C 180,E1 -2544.249,E2 -2544.249} C_VEL
LIN {X 0,Y 696.387,Z 198.477,A -85,B 0,C 180,E1 -2547.168,E2 -2547.168} C_VEL
LIN {X 0,Y 696.368,Z 198.487,A -85,B 0,C 180,E1 -2550.264,E2 -2550.264} C_VEL
LIN {X 0,Y 696.37,Z 198.482,A -85,B 0,C 180,E1 -2553.068,E2 -2553.068} C_VEL
LIN {X 0,Y 696.373,Z 198.489,A -85,B 0,C 180,E1 -2556.201,E2 -2556.201} C_VEL
LIN {X 0,Y 696.356,Z 198.484,A -85,B 0,C 180,E1 -2558.971,E2 -2558.971} C_VEL
LIN {X 0,Y 696.395,Z 198.486,A -85,B 0,C 180,E1 -2561.997,E2 -2561.997} C_VEL
LIN {X 0,Y 696.344,Z 198.486,A -85,B 0,C 180,E1 -2564.833,E2 -2564.833} C_VEL
LIN {X 0,Y 696.405,Z 198.488,A -85,B 0,C 180,E1 -2567.683,E2 -2567.683} C_VEL
LIN {X 0,Y 696.35,Z 198.557,A -85,B 0,C 180,E1 -2568.717,E2 -2568.717} C_VEL
LIN {X 0,Y 697.377,Z 201.538,A -85,B 0,C 180,E1 -2568.953,E2 -2568.953} C_VEL
LIN {X 0,Y 700.476,Z 207.638,A -85,B 0,C 180,E1 -2569.497,E2 -2569.497} C_VEL
LIN {X 0,Y 706.642,Z 220.935,A -85,B 0,C 180,E1 -2570.572,E2 -2570.572} C_VEL
LIN {X 0,Y 705.501,Z 275.624,A -85,B 0,C 180,E1 -2573.165,E2 -2573.165} C_VEL
LIN {X 0,Y 705.077,Z 299.347,A -85,B 0,C 180,E1 -2574.253,E2 -2574.253} C_VEL
LIN {X 0,Y 706.723,Z 311.115,A -85,B 0,C 180,E1 -2574.493,E2 -2574.493} C_VEL
LIN {X 0,Y 704.97,Z 577.177,A -85,B 0,C 180,E1 -2577.594,E2 -2577.594} C_VEL
LIN {X 0,Y 704.209,Z 691.357,A -85,B 0,C 180,E1 -2578.922,E2 -2578.922} C_VEL
LIN {X 0,Y 703.76,Z 716.892,A -85,B 0,C 180,E1 -2579.368,E2 -2579.368} C_VEL
LIN {X 0,Y 703.262,Z 738.672,A -85,B 0,C 180,E1 -2579.884,E2 -2579.884} C_VEL
LIN {X 0,Y 702.682,Z 762.561,A -85,B 0,C 180,E1 -2580.599,E2 -2580.599} C_VEL
LIN {X 0,Y 702.004,Z 784.489,A -85,B 0,C 180,E1 -2581.407,E2 -2581.407} C_VEL
LIN {X 0,Y 701.295,Z 807.166,A -85,B 0,C 180,E1 -2582.395,E2 -2582.395} C_VEL
LIN {X 0,Y 700.533,Z 828.597,A -85,B 0,C 180,E1 -2583.501,E2 -2583.501} C_VEL
LIN {X 0,Y 699.773,Z 849.761,A -85,B 0,C 180,E1 -2584.754,E2 -2584.754} C_VEL
LIN {X 0,Y 699.088,Z 868.771,A -85,B 0,C 180,E1 -2586.057,E2 -2586.057} C_VEL
LIN {X 0,Y 698.419,Z 887.762,A -85,B 0,C 180,E1 -2587.527,E2 -2587.527} C_VEL
LIN {X 0,Y 697.857,Z 904.463,A -85,B 0,C 180,E1 -2589.01,E2 -2589.01} C_VEL
LIN {X 0,Y 697.329,Z 920.969,A -85,B 0,C 180,E1 -2590.657,E2 -2590.657} C_VEL
LIN {X 0,Y 696.899,Z 935.933,A -85,B 0,C 180,E1 -2592.378,E2 -2592.378} C_VEL
LIN {X 0,Y 696.577,Z 949.644,A -85,B 0,C 180,E1 -2594.173,E2 -2594.173} C_VEL
LIN {X 0,Y 696.33,Z 961.319,A -85,B 0,C 180,E1 -2595.956,E2 -2595.956} C_VEL
LIN {X 0,Y 696.151,Z 972.299,A -85,B 0,C 180,E1 -2597.895,E2 -2597.895} C_VEL
LIN {X 0,Y 696.03,Z 981.25,A -85,B 0,C 180,E1 -2599.823,E2 -2599.823} C_VEL
LIN {X 0,Y 695.956,Z 988.333,A -85,B 0,C 180,E1 -2601.656,E2 -2601.656} C_VEL
LIN {X 0,Y 695.919,Z 994.277,A -85,B 0,C 180,E1 -2603.648,E2 -2603.648} C_VEL
LIN {X 0,Y 695.917,Z 998.132,A -85,B 0,C 180,E1 -2605.385,E2 -2605.385} C_VEL
LIN {X 0,Y 695.888,Z 1001.092,A -85,B 0,C 180,E1 -2607.365,E2 -2607.365} C_VEL
LIN {X 0,Y 695.885,Z 1002.306,A -85,B 0,C 180,E1 -2609.259,E2 -2609.259} C_VEL
LIN {X 0,Y 695.899,Z 1002.239,A -85,B 0,C 180,E1 -2610.988,E2 -2610.988} C_VEL
LIN {X 0,Y 695.885,Z 1000.573,A -85,B 0,C 180,E1 -2613.048,E2 -2613.048} C_VEL
LIN {X 0,Y 695.906,Z 997.814,A -85,B 0,C 180,E1 -2614.78,E2 -2614.78} C_VEL
LIN {X 0,Y 695.932,Z 993.244,A -85,B 0,C 180,E1 -2616.766,E2 -2616.766} C_VEL
LIN {X 0,Y 695.946,Z 987.014,A -85,B 0,C 180,E1 -2618.706,E2 -2618.706} C_VEL
LIN {X 0,Y 696.047,Z 980.184,A -85,B 0,C 180,E1 -2620.428,E2 -2620.428} C_VEL
LIN {X 0,Y 696.181,Z 970.03,A -85,B 0,C 180,E1 -2622.526,E2 -2622.526} C_VEL
LIN {X 0,Y 696.357,Z 960.057,A -85,B 0,C 180,E1 -2624.25,E2 -2624.25} C_VEL
LIN {X 0,Y 696.635,Z 946.833,A -85,B 0,C 180,E1 -2626.213,E2 -2626.213} C_VEL
LIN {X 0,Y 696.969,Z 933.81,A -85,B 0,C 180,E1 -2627.879,E2 -2627.879} C_VEL
LIN {X 0,Y 697.43,Z 917.639,A -85,B 0,C 180,E1 -2629.689,E2 -2629.689} C_VEL
LIN {X 0,Y 697.916,Z 902.605,A -85,B 0,C 180,E1 -2631.164,E2 -2631.164} C_VEL
LIN {X 0,Y 698.559,Z 883.396,A -85,B 0,C 180,E1 -2632.824,E2 -2632.824} C_VEL
LIN {X 0,Y 699.193,Z 865.728,A -85,B 0,C 180,E1 -2634.163,E2 -2634.163} C_VEL
LIN {X 0,Y 699.955,Z 844.715,A -85,B 0,C 180,E1 -2635.557,E2 -2635.557} C_VEL
LIN {X 0,Y 700.618,Z 826.323,A -85,B 0,C 180,E1 -2636.624,E2 -2636.624} C_VEL
LIN {X 0,Y 701.397,Z 803.26,A -85,B 0,C 180,E1 -2637.785,E2 -2637.785} C_VEL
LIN {X 0,Y 702.081,Z 782.227,A -85,B 0,C 180,E1 -2638.682,E2 -2638.682} C_VEL
LIN {X 0,Y 702.779,Z 759.174,A -85,B 0,C 180,E1 -2639.514,E2 -2639.514} C_VEL
LIN {X 0,Y 703.313,Z 736.186,A -85,B 0,C 180,E1 -2640.181,E2 -2640.181} C_VEL
LIN {X 0,Y 703.913,Z 712.037,A -85,B 0,C 180,E1 -2640.734,E2 -2640.734} C_VEL
LIN {X 0,Y 704.23,Z 688.169,A -85,B 0,C 180,E1 -2641.121,E2 -2641.121} C_VEL
LIN {X 0,Y 705.761,Z 447.928,A -85,B 0,C 180,E1 -2643.904,E2 -2643.904} C_VEL
LIN {X 0,Y 706.574,Z 308.693,A -85,B 0,C 180,E1 -2645.546,E2 -2645.546} C_VEL
LIN {X 0,Y 704.965,Z 298.307,A -85,B 0,C 180,E1 -2645.777,E2 -2645.777} C_VEL
LIN {X 0,Y 706.162,Z 241.411,A -85,B 0,C 180,E1 -2648.433,E2 -2648.433} C_VEL
LIN {X 0,Y 706.508,Z 220.477,A -85,B 0,C 180,E1 -2649.438,E2 -2649.438} C_VEL
LIN {X 0,Y 699.556,Z 205.772,A -85,B 0,C 180,E1 -2650.752,E2 -2650.752} C_VEL
LIN {X 0,Y 697.91,Z 202.316,A -85,B 0,C 180,E1 -2651.097,E2 -2651.097} C_VEL
LIN {X 0,Y 696.412,Z 198.761,A -85,B 0,C 180,E1 -2651.455,E2 -2651.455} C_VEL
LIN {X 0,Y 696.394,Z 198.489,A -85,B 0,C 180,E1 -2651.701,E2 -2651.701} C_VEL
LIN {X 0,Y 696.4,Z 198.489,A -85,B 0,C 180,E1 -2654.712,E2 -2654.712} C_VEL
LIN {X 0,Y 696.399,Z 198.488,A -85,B 0,C 180,E1 -2657.684,E2 -2657.684} C_VEL
LIN {X 0,Y 696.389,Z 198.489,A -85,B 0,C 180,E1 -2660.713,E2 -2660.713} C_VEL
LIN {X 0,Y 696.38,Z 198.49,A -85,B 0,C 180,E1 -2663.659,E2 -2663.659} C_VEL
LIN {X 0,Y 696.412,Z 198.548,A -85,B 0,C 180,E1 -2664.601,E2 -2664.601} C_VEL
LIN {X 0,Y 697.568,Z 201.776,A -85,B 0,C 180,E1 -2664.932,E2 -2664.932} C_VEL
LIN {X 0,Y 702.995,Z 214.863,A -85,B 0,C 180,E1 -2666.231,E2 -2666.231} C_VEL
LIN {X 0,Y 703.618,Z 217.425,A -85,B 0,C 180,E1 -2666.441,E2 -2666.441} C_VEL
LIN {X 0,Y 701.761,Z 265.146,A -85,B 0,C 180,E1 -2669.33,E2 -2669.33} C_VEL
LIN {X 0,Y 700.403,Z 322.039,A -85,B 0,C 180,E1 -2672.619,E2 -2672.619} C_VEL
LIN {X 0,Y 699.523,Z 375.312,A -85,B 0,C 180,E1 -2675.601,E2 -2675.601} C_VEL
LIN {X 0,Y 698.765,Z 430.143,A -85,B 0,C 180,E1 -2678.599,E2 -2678.599} C_VEL
LIN {X 0,Y 698.363,Z 465.064,A -85,B 0,C 180,E1 -2680.46,E2 -2680.46} C_VEL
LIN {X 0,Y 699.86,Z 478.846,A -85,B 0,C 180,E1 -2680.693,E2 -2680.693} C_VEL
LIN {X 0,Y 698.784,Z 614.753,A -85,B 0,C 180,E1 -2682.236,E2 -2682.236} C_VEL
LIN {X 0,Y 698.463,Z 681.133,A -85,B 0,C 180,E1 -2682.989,E2 -2682.989} C_VEL
LIN {X 0,Y 698.264,Z 700.156,A -85,B 0,C 180,E1 -2683.358,E2 -2683.358} C_VEL
LIN {X 0,Y 698.014,Z 718.42,A -85,B 0,C 180,E1 -2683.865,E2 -2683.865} C_VEL
LIN {X 0,Y 697.708,Z 735.718,A -85,B 0,C 180,E1 -2684.498,E2 -2684.498} C_VEL
LIN {X 0,Y 697.411,Z 752.149,A -85,B 0,C 180,E1 -2685.257,E2 -2685.257} C_VEL
LIN {X 0,Y 697.096,Z 767.73,A -85,B 0,C 180,E1 -2686.141,E2 -2686.141} C_VEL
LIN {X 0,Y 696.804,Z 782.562,A -85,B 0,C 180,E1 -2687.149,E2 -2687.149} C_VEL
LIN {X 0,Y 696.55,Z 795.949,A -85,B 0,C 180,E1 -2688.239,E2 -2688.239} C_VEL
LIN {X 0,Y 696.327,Z 808.765,A -85,B 0,C 180,E1 -2689.492,E2 -2689.492} C_VEL
LIN {X 0,Y 696.159,Z 820.017,A -85,B 0,C 180,E1 -2690.826,E2 -2690.826} C_VEL
LIN {X 0,Y 696.042,Z 829.727,A -85,B 0,C 180,E1 -2692.239,E2 -2692.239} C_VEL
LIN {X 0,Y 695.969,Z 837.458,A -85,B 0,C 180,E1 -2693.649,E2 -2693.649} C_VEL
LIN {X 0,Y 695.935,Z 843.749,A -85,B 0,C 180,E1 -2695.137,E2 -2695.137} C_VEL
LIN {X 0,Y 695.914,Z 848.47,A -85,B 0,C 180,E1 -2696.705,E2 -2696.705} C_VEL
LIN {X 0,Y 695.914,Z 851.344,A -85,B 0,C 180,E1 -2698.271,E2 -2698.271} C_VEL
LIN {X 0,Y 695.915,Z 852.45,A -85,B 0,C 180,E1 -2699.835,E2 -2699.835} C_VEL
LIN {X 0,Y 695.911,Z 851.815,A -85,B 0,C 180,E1 -2701.4,E2 -2701.4} C_VEL
LIN {X 0,Y 695.918,Z 849.429,A -85,B 0,C 180,E1 -2702.965,E2 -2702.965} C_VEL
LIN {X 0,Y 695.927,Z 845.48,A -85,B 0,C 180,E1 -2704.45,E2 -2704.45} C_VEL
LIN {X 0,Y 695.953,Z 839.807,A -85,B 0,C 180,E1 -2705.938,E2 -2705.938} C_VEL
LIN {X 0,Y 696.016,Z 832.713,A -85,B 0,C 180,E1 -2707.346,E2 -2707.346} C_VEL
LIN {X 0,Y 696.111,Z 823.748,A -85,B 0,C 180,E1 -2708.758,E2 -2708.758} C_VEL
LIN {X 0,Y 696.26,Z 813.325,A -85,B 0,C 180,E1 -2710.091,E2 -2710.091} C_VEL
LIN {X 0,Y 696.453,Z 801.453,A -85,B 0,C 180,E1 -2711.344,E2 -2711.344} C_VEL
LIN {X 0,Y 696.7,Z 788.1,A -85,B 0,C 180,E1 -2712.516,E2 -2712.516} C_VEL
LIN {X 0,Y 696.992,Z 773.136,A -85,B 0,C 180,E1 -2713.608,E2 -2713.608} C_VEL
LIN {X 0,Y 697.307,Z 757.411,A -85,B 0,C 180,E1 -2714.555,E2 -2714.555} C_VEL
LIN {X 0,Y 697.602,Z 740.74,A -85,B 0,C 180,E1 -2715.377,E2 -2715.377} C_VEL
LIN {X 0,Y 697.929,Z 723.561,A -85,B 0,C 180,E1 -2716.052,E2 -2716.052} C_VEL
LIN {X 0,Y 698.192,Z 705.148,A -85,B 0,C 180,E1 -2716.607,E2 -2716.607} C_VEL
LIN {X 0,Y 698.405,Z 686.432,A -85,B 0,C 180,E1 -2717.01,E2 -2717.01} C_VEL
LIN {X 0,Y 698.554,Z 664.873,A -85,B 0,C 180,E1 -2717.3,E2 -2717.3} C_VEL
LIN {X 0,Y 698.559,Z 663.716,A -85,B 0,C 180,E1 -2717.312,E2 -2717.312} C_VEL
LIN {X 0,Y 697.628,Z 656.12,A -85,B 0,C 180,E1 -2717.422,E2 -2717.422} C_VEL
LIN {X 0,Y 691.754,Z 636.216,A -85,B 0,C 180,E1 -2717.799,E2 -2717.799} C_VEL
LIN {X 0,Y 691.079,Z 629.682,A -85,B 0,C 180,E1 -2717.888,E2 -2717.888} C_VEL
LIN {X 0,Y 691.757,Z 476.22,A -85,B 0,C 180,E1 -2719.585,E2 -2719.585} C_VEL
LIN {X 0,Y 690.687,Z 467.362,A -85,B 0,C 180,E1 -2719.735,E2 -2719.735} C_VEL
LIN {X 0,Y 691.604,Z 411.541,A -85,B 0,C 180,E1 -2722.797,E2 -2722.797} C_VEL
LIN {X 0,Y 692.526,Z 357.73,A -85,B 0,C 180,E1 -2725.806,E2 -2725.806} C_VEL
LIN {X 0,Y 693.468,Z 308.718,A -85,B 0,C 180,E1 -2728.586,E2 -2728.586} C_VEL
LIN {X 0,Y 694.686,Z 254.271,A -85,B 0,C 180,E1 -2731.736,E2 -2731.736} C_VEL
LIN {X 0,Y 695.434,Z 218.314,A -85,B 0,C 180,E1 -2733.86,E2 -2733.86} C_VEL
LIN {X 0,Y 688.466,Z 199.475,A -85,B 0,C 180,E1 -2735.415,E2 -2735.415} C_VEL
LIN {X 0,Y 688.413,Z 199.479,A -85,B 0,C 180,E1 -2738.341,E2 -2738.341} C_VEL
LIN {X 0,Y 688.459,Z 199.476,A -85,B 0,C 180,E1 -2741.252,E2 -2741.252} C_VEL
LIN {X 0,Y 688.43,Z 199.476,A -85,B 0,C 180,E1 -2744.2,E2 -2744.2} C_VEL
LIN {X 0,Y 688.441,Z 199.472,A -85,B 0,C 180,E1 -2747.064,E2 -2747.064} C_VEL
LIN {X 0,Y 688.433,Z 199.478,A -85,B 0,C 180,E1 -2750.074,E2 -2750.074} C_VEL
LIN {X 0,Y 688.409,Z 199.483,A -85,B 0,C 180,E1 -2752.883,E2 -2752.883} C_VEL
LIN {X 0,Y 688.456,Z 199.683,A -85,B 0,C 180,E1 -2753.97,E2 -2753.97} C_VEL
LIN {X 0,Y 694.615,Z 216.106,A -85,B 0,C 180,E1 -2755.499,E2 -2755.499} C_VEL
LIN {X 0,Y 695.816,Z 220.075,A -85,B 0,C 180,E1 -2755.865,E2 -2755.865} C_VEL
LIN {X 0,Y 694.796,Z 259.327,A -85,B 0,C 180,E1 -2758.7,E2 -2758.7} C_VEL
LIN {X 0,Y 693.822,Z 286.378,A -85,B 0,C 180,E1 -2760.679,E2 -2760.679} C_VEL
LIN {X 0,Y 693.028,Z 305.154,A -85,B 0,C 180,E1 -2762.069,E2 -2762.069} C_VEL
LIN {X 0,Y 695.332,Z 317.607,A -85,B 0,C 180,E1 -2762.312,E2 -2762.312} C_VEL
LIN {X 0,Y 693.715,Z 603.355,A -85,B 0,C 180,E1 -2765.488,E2 -2765.488} C_VEL
LIN {X 0,Y 693.473,Z 621.628,A -85,B 0,C 180,E1 -2765.776,E2 -2765.776} C_VEL
LIN {X 0,Y 693.136,Z 640.087,A -85,B 0,C 180,E1 -2766.177,E2 -2766.177} C_VEL
LIN {X 0,Y 692.732,Z 658.203,A -85,B 0,C 180,E1 -2766.681,E2 -2766.681} C_VEL
LIN {X 0,Y 692.239,Z 679.129,A -85,B 0,C 180,E1 -2767.405,E2 -2767.405} C_VEL
LIN {X 0,Y 691.651,Z 699.38,A -85,B 0,C 180,E1 -2768.279,E2 -2768.279} C_VEL
LIN {X 0,Y 691.114,Z 716.765,A -85,B 0,C 180,E1 -2769.168,E2 -2769.168} C_VEL
LIN {X 0,Y 690.586,Z 733.368,A -85,B 0,C 180,E1 -2770.152,E2 -2770.152} C_VEL
LIN {X 0,Y 690.055,Z 750.457,A -85,B 0,C 180,E1 -2771.323,E2 -2771.323} C_VEL
LIN {X 0,Y 689.512,Z 768.174,A -85,B 0,C 180,E1 -2772.749,E2 -2772.749} C_VEL
LIN {X 0,Y 689.083,Z 782.384,A -85,B 0,C 180,E1 -2774.083,E2 -2774.083} C_VEL
LIN {X 0,Y 688.746,Z 795.167,A -85,B 0,C 180,E1 -2775.454,E2 -2775.454} C_VEL
LIN {X 0,Y 688.435,Z 808.796,A -85,B 0,C 180,E1 -2777.161,E2 -2777.161} C_VEL
LIN {X 0,Y 688.217,Z 819.525,A -85,B 0,C 180,E1 -2778.774,E2 -2778.774} C_VEL
LIN {X 0,Y 688.086,Z 828.13,A -85,B 0,C 180,E1 -2780.296,E2 -2780.296} C_VEL
LIN {X 0,Y 688.002,Z 836.002,A -85,B 0,C 180,E1 -2781.98,E2 -2781.98} C_VEL
LIN {X 0,Y 687.938,Z 843.277,A -85,B 0,C 180,E1 -2783.993,E2 -2783.993} C_VEL
LIN {X 0,Y 687.923,Z 847.67,A -85,B 0,C 180,E1 -2785.665,E2 -2785.665} C_VEL
LIN {X 0,Y 687.912,Z 850.609,A -85,B 0,C 180,E1 -2787.334,E2 -2787.334} C_VEL
LIN {X 0,Y 687.914,Z 852.301,A -85,B 0,C 180,E1 -2789.167,E2 -2789.167} C_VEL
LIN {X 0,Y 687.907,Z 852.2,A -85,B 0,C 180,E1 -2791.083,E2 -2791.083} C_VEL
LIN {X 0,Y 687.909,Z 850.5,A -85,B 0,C 180,E1 -2792.833,E2 -2792.833} C_VEL
LIN {X 0,Y 687.919,Z 847.327,A -85,B 0,C 180,E1 -2794.585,E2 -2794.585} C_VEL
LIN {X 0,Y 687.942,Z 842.019,A -85,B 0,C 180,E1 -2796.51,E2 -2796.51} C_VEL
LIN {X 0,Y 688.006,Z 835.314,A -85,B 0,C 180,E1 -2798.272,E2 -2798.272} C_VEL
LIN {X 0,Y 688.101,Z 827.283,A -85,B 0,C 180,E1 -2799.958,E2 -2799.958} C_VEL
LIN {X 0,Y 688.263,Z 817.487,A -85,B 0,C 180,E1 -2801.65,E2 -2801.65} C_VEL
LIN {X 0,Y 688.502,Z 805.631,A -85,B 0,C 180,E1 -2803.351,E2 -2803.351} C_VEL
LIN {X 0,Y 688.804,Z 792.928,A -85,B 0,C 180,E1 -2804.888,E2 -2804.888} C_VEL
LIN {X 0,Y 689.152,Z 779.852,A -85,B 0,C 180,E1 -2806.262,E2 -2806.262} C_VEL
LIN {X 0,Y 689.655,Z 763.188,A -85,B 0,C 180,E1 -2807.77,E2 -2807.77} C_VEL
LIN {X 0,Y 690.162,Z 746.849,A -85,B 0,C 180,E1 -2809.025,E2 -2809.025} C_VEL
LIN {X 0,Y 690.671,Z 730.636,A -85,B 0,C 180,E1 -2810.11,E2 -2810.11} C_VEL
LIN {X 0,Y 691.266,Z 712.545,A -85,B 0,C 180,E1 -2811.155,E2 -2811.155} C_VEL
LIN {X 0,Y 691.877,Z 691.767,A -85,B 0,C 180,E1 -2812.16,E2 -2812.16} C_VEL
LIN {X 0,Y 692.376,Z 673.27,A -85,B 0,C 180,E1 -2812.9,E2 -2812.9} C_VEL
LIN {X 0,Y 692.771,Z 656.015,A -85,B 0,C 180,E1 -2813.475,E2 -2813.475} C_VEL
LIN {X 0,Y 693.178,Z 638.161,A -85,B 0,C 180,E1 -2813.96,E2 -2813.96} C_VEL
LIN {X 0,Y 693.52,Z 618.807,A -85,B 0,C 180,E1 -2814.367,E2 -2814.367} C_VEL
LIN {X 0,Y 693.807,Z 595.213,A -85,B 0,C 180,E1 -2814.706,E2 -2814.706} C_VEL
LIN {X 0,Y 695.329,Z 316.439,A -85,B 0,C 180,E1 -2817.791,E2 -2817.791} C_VEL
LIN {X 0,Y 692.953,Z 304.605,A -85,B 0,C 180,E1 -2818.039,E2 -2818.039} C_VEL
LIN {X 0,Y 694.338,Z 274.175,A -85,B 0,C 180,E1 -2820.314,E2 -2820.314} C_VEL
LIN {X 0,Y 695.424,Z 236.86,A -85,B 0,C 180,E1 -2823.02,E2 -2823.02} C_VEL
LIN {X 0,Y 695.747,Z 219.344,A -85,B 0,C 180,E1 -2824.289,E2 -2824.289} C_VEL
LIN {X 0,Y 689.56,Z 202.639,A -85,B 0,C 180,E1 -2825.861,E2 -2825.861} C_VEL
LIN {X 0,Y 688.459,Z 199.475,A -85,B 0,C 180,E1 -2826.146,E2 -2826.146} C_VEL
LIN {X 0,Y 688.43,Z 199.477,A -85,B 0,C 180,E1 -2829.076,E2 -2829.076} C_VEL
LIN {X 0,Y 688.456,Z 199.475,A -85,B 0,C 180,E1 -2832.032,E2 -2832.032} C_VEL
LIN {X 0,Y 688.434,Z 199.474,A -85,B 0,C 180,E1 -2835.018,E2 -2835.018} C_VEL
LIN {X 0,Y 688.455,Z 199.476,A -85,B 0,C 180,E1 -2837.968,E2 -2837.968} C_VEL
LIN {X 0,Y 688.44,Z 199.47,A -85,B 0,C 180,E1 -2840.924,E2 -2840.924} C_VEL
LIN {X 0,Y 688.459,Z 199.474,A -85,B 0,C 180,E1 -2843.867,E2 -2843.867} C_VEL
LIN {X 0,Y 688.446,Z 199.464,A -85,B 0,C 180,E1 -2846.932,E2 -2846.932} C_VEL
LIN {X 0,Y 688.455,Z 199.472,A -85,B 0,C 180,E1 -2849.929,E2 -2849.929} C_VEL
LIN {X 0,Y 688.449,Z 199.466,A -85,B 0,C 180,E1 -2852.961,E2 -2852.961} C_VEL
LIN {X 0,Y 688.452,Z 199.465,A -85,B 0,C 180,E1 -2856,E2 -2856} C_VEL
LIN {X 0,Y 688.454,Z 199.467,A -85,B 0,C 180,E1 -2858.977,E2 -2858.977} C_VEL
LIN {X 0,Y 688.451,Z 199.466,A -85,B 0,C 180,E1 -2861.979,E2 -2861.979} C_VEL
LIN {X 0,Y 688.456,Z 199.467,A -85,B 0,C 180,E1 -2865.018,E2 -2865.018} C_VEL
LIN {X 0,Y 688.449,Z 199.467,A -85,B 0,C 180,E1 -2868.013,E2 -2868.013} C_VEL
LIN {X 0,Y 688.458,Z 199.467,A -85,B 0,C 180,E1 -2871.06,E2 -2871.06} C_VEL
LIN {X 0,Y 688.444,Z 199.466,A -85,B 0,C 180,E1 -2874.081,E2 -2874.081} C_VEL
LIN {X 0,Y 688.46,Z 199.467,A -85,B 0,C 180,E1 -2877.086,E2 -2877.086} C_VEL
LIN {X 0,Y 688.444,Z 199.463,A -85,B 0,C 180,E1 -2880.083,E2 -2880.083} C_VEL
LIN {X 0,Y 688.461,Z 199.466,A -85,B 0,C 180,E1 -2883.08,E2 -2883.08} C_VEL
LIN {X 0,Y 688.437,Z 199.464,A -85,B 0,C 180,E1 -2886.17,E2 -2886.17} C_VEL
LIN {X 0,Y 688.464,Z 199.464,A -85,B 0,C 180,E1 -2889.193,E2 -2889.193} C_VEL
LIN {X 0,Y 688.433,Z 199.474,A -85,B 0,C 180,E1 -2892.243,E2 -2892.243} C_VEL
LIN {X 0,Y 688.467,Z 199.466,A -85,B 0,C 180,E1 -2895.241,E2 -2895.241} C_VEL
LIN {X 0,Y 688.429,Z 199.473,A -85,B 0,C 180,E1 -2898.284,E2 -2898.284} C_VEL
LIN {X 0,Y 688.461,Z 199.467,A -85,B 0,C 180,E1 -2901.201,E2 -2901.201} C_VEL
LIN {X 0,Y 688.43,Z 199.475,A -85,B 0,C 180,E1 -2904.27,E2 -2904.27} C_VEL
LIN {X 0,Y 688.454,Z 199.466,A -85,B 0,C 180,E1 -2907.226,E2 -2907.226} C_VEL
LIN {X 0,Y 688.429,Z 199.477,A -85,B 0,C 180,E1 -2910.265,E2 -2910.265} C_VEL
LIN {X 0,Y 688.434,Z 199.471,A -85,B 0,C 180,E1 -2913.101,E2 -2913.101} C_VEL
LIN {X 0,Y 688.431,Z 199.478,A -85,B 0,C 180,E1 -2916.238,E2 -2916.238} C_VEL
LIN {X 0,Y 688.425,Z 199.472,A -85,B 0,C 180,E1 -2919.077,E2 -2919.077} C_VEL
LIN {X 0,Y 688.435,Z 199.479,A -85,B 0,C 180,E1 -2922.206,E2 -2922.206} C_VEL
LIN {X 0,Y 688.411,Z 199.474,A -85,B 0,C 180,E1 -2924.98,E2 -2924.98} C_VEL
LIN {X 0,Y 688.462,Z 199.478,A -85,B 0,C 180,E1 -2927.969,E2 -2927.969} C_VEL
LIN {X 0,Y 688.45,Z 199.58,A -85,B 0,C 180,E1 -2928.192,E2 -2928.192} C_VEL
LIN {X 0,Y 689.516,Z 202.648,A -85,B 0,C 180,E1 -2928.441,E2 -2928.441} C_VEL
LIN {X 0,Y 696.062,Z 215.958,A -85,B 0,C 180,E1 -2929.62,E2 -2929.62} C_VEL
LIN {X 0,Y 700.012,Z 224.6,A -85,B 0,C 180,E1 -2930.321,E2 -2930.321} C_VEL
LIN {X 0,Y 698.681,Z 280.566,A -85,B 0,C 180,E1 -2932.993,E2 -2932.993} C_VEL
LIN {X 0,Y 698.335,Z 299.337,A -85,B 0,C 180,E1 -2933.853,E2 -2933.853} C_VEL
LIN {X 0,Y 700.196,Z 312.407,A -85,B 0,C 180,E1 -2934.127,E2 -2934.127} C_VEL
LIN {X 0,Y 698.195,Z 579.722,A -85,B 0,C 180,E1 -2937.271,E2 -2937.271} C_VEL
LIN {X 0,Y 697.348,Z 691.401,A -85,B 0,C 180,E1 -2938.583,E2 -2938.583} C_VEL
LIN {X 0,Y 696.858,Z 716.759,A -85,B 0,C 180,E1 -2939.028,E2 -2939.028} C_VEL
LIN {X 0,Y 696.284,Z 738.562,A -85,B 0,C 180,E1 -2939.547,E2 -2939.547} C_VEL
LIN {X 0,Y 695.63,Z 762.557,A -85,B 0,C 180,E1 -2940.271,E2 -2940.271} C_VEL
LIN {X 0,Y 694.911,Z 783.354,A -85,B 0,C 180,E1 -2941.041,E2 -2941.041} C_VEL
LIN {X 0,Y 694.117,Z 805.252,A -85,B 0,C 180,E1 -2941.991,E2 -2941.991} C_VEL
LIN {X 0,Y 693.259,Z 827.137,A -85,B 0,C 180,E1 -2943.118,E2 -2943.118} C_VEL
LIN {X 0,Y 692.489,Z 846.179,A -85,B 0,C 180,E1 -2944.239,E2 -2944.239} C_VEL
LIN {X 0,Y 691.611,Z 867.23,A -85,B 0,C 180,E1 -2945.667,E2 -2945.667} C_VEL
LIN {X 0,Y 690.896,Z 885.056,A -85,B 0,C 180,E1 -2947.044,E2 -2947.044} C_VEL
LIN {X 0,Y 690.213,Z 902.605,A -85,B 0,C 180,E1 -2948.588,E2 -2948.588} C_VEL
LIN {X 0,Y 689.669,Z 917.638,A -85,B 0,C 180,E1 -2950.08,E2 -2950.08} C_VEL
LIN {X 0,Y 689.134,Z 933.813,A -85,B 0,C 180,E1 -2951.911,E2 -2951.911} C_VEL
LIN {X 0,Y 688.759,Z 946.529,A -85,B 0,C 180,E1 -2953.556,E2 -2953.556} C_VEL
LIN {X 0,Y 688.438,Z 959.761,A -85,B 0,C 180,E1 -2955.534,E2 -2955.534} C_VEL
LIN {X 0,Y 688.231,Z 969.568,A -85,B 0,C 180,E1 -2957.242,E2 -2957.242} C_VEL
LIN {X 0,Y 688.063,Z 979.475,A -85,B 0,C 180,E1 -2959.28,E2 -2959.28} C_VEL
LIN {X 0,Y 687.966,Z 986.513,A -85,B 0,C 180,E1 -2961.053,E2 -2961.053} C_VEL
LIN {X 0,Y 687.931,Z 992.253,A -85,B 0,C 180,E1 -2962.819,E2 -2962.819} C_VEL
LIN {X 0,Y 687.891,Z 997.338,A -85,B 0,C 180,E1 -2964.913,E2 -2964.913} C_VEL
LIN {X 0,Y 687.903,Z 1000.236,A -85,B 0,C 180,E1 -2966.667,E2 -2966.667} C_VEL
LIN {X 0,Y 687.91,Z 1002.171,A -85,B 0,C 180,E1 -2968.751,E2 -2968.751} C_VEL
LIN {X 0,Y 687.882,Z 1002.351,A -85,B 0,C 180,E1 -2970.583,E2 -2970.583} C_VEL
LIN {X 0,Y 687.905,Z 1001.296,A -85,B 0,C 180,E1 -2972.416,E2 -2972.416} C_VEL
LIN {X 0,Y 687.918,Z 998.448,A -85,B 0,C 180,E1 -2974.502,E2 -2974.502} C_VEL
LIN {X 0,Y 687.924,Z 994.689,A -85,B 0,C 180,E1 -2976.258,E2 -2976.258} C_VEL
LIN {X 0,Y 687.973,Z 989.148,A -85,B 0,C 180,E1 -2978.206,E2 -2978.206} C_VEL
LIN {X 0,Y 688.046,Z 981.605,A -85,B 0,C 180,E1 -2980.212,E2 -2980.212} C_VEL
LIN {X 0,Y 688.162,Z 973.524,A -85,B 0,C 180,E1 -2981.992,E2 -2981.992} C_VEL
LIN {X 0,Y 688.375,Z 962.356,A -85,B 0,C 180,E1 -2984.039,E2 -2984.039} C_VEL
LIN {X 0,Y 688.624,Z 951.385,A -85,B 0,C 180,E1 -2985.755,E2 -2985.755} C_VEL
LIN {X 0,Y 689.012,Z 937.332,A -85,B 0,C 180,E1 -2987.656,E2 -2987.656} C_VEL
LIN {X 0,Y 689.463,Z 923.3,A -85,B 0,C 180,E1 -2989.309,E2 -2989.309} C_VEL
LIN {X 0,Y 690.089,Z 906.16,A -85,B 0,C 180,E1 -2991.074,E2 -2991.074} C_VEL
LIN {X 0,Y 690.7,Z 889.787,A -85,B 0,C 180,E1 -2992.559,E2 -2992.559} C_VEL
LIN {X 0,Y 691.496,Z 870.26,A -85,B 0,C 180,E1 -2994.11,E2 -2994.11} C_VEL
LIN {X 0,Y 692.24,Z 851.743,A -85,B 0,C 180,E1 -2995.404,E2 -2995.404} C_VEL
LIN {X 0,Y 693.127,Z 830.364,A -85,B 0,C 180,E1 -2996.703,E2 -2996.703} C_VEL
LIN {X 0,Y 693.907,Z 810.763,A -85,B 0,C 180,E1 -2997.738,E2 -2997.738} C_VEL
LIN {X 0,Y 694.788,Z 786.736,A -85,B 0,C 180,E1 -2998.823,E2 -2998.823} C_VEL
LIN {X 0,Y 695.479,Z 766.409,A -85,B 0,C 180,E1 -2999.594,E2 -2999.594} C_VEL
LIN {X 0,Y 696.232,Z 741.99,A -85,B 0,C 180,E1 -3000.361,E2 -3000.361} C_VEL
LIN {X 0,Y 696.762,Z 719.611,A -85,B 0,C 180,E1 -3000.911,E2 -3000.911} C_VEL
LIN {X 0,Y 697.321,Z 695.022,A -85,B 0,C 180,E1 -3001.368,E2 -3001.368} C_VEL
LIN {X 0,Y 697.718,Z 648.066,A -85,B 0,C 180,E1 -3001.938,E2 -3001.938} C_VEL
LIN {X 0,Y 699.507,Z 400.707,A -85,B 0,C 180,E1 -3004.825,E2 -3004.825} C_VEL
LIN {X 0,Y 700.021,Z 309.905,A -85,B 0,C 180,E1 -3005.915,E2 -3005.915} C_VEL
LIN {X 0,Y 698.228,Z 298.171,A -85,B 0,C 180,E1 -3006.183,E2 -3006.183} C_VEL
LIN {X 0,Y 699.098,Z 250.456,A -85,B 0,C 180,E1 -3008.392,E2 -3008.392} C_VEL
LIN {X 0,Y 699.861,Z 224.104,A -85,B 0,C 180,E1 -3009.69,E2 -3009.69} C_VEL
LIN {X 0,Y 693.919,Z 211.305,A -85,B 0,C 180,E1 -3010.858,E2 -3010.858} C_VEL
LIN {X 0,Y 689.985,Z 203.273,A -85,B 0,C 180,E1 -3011.728,E2 -3011.728} C_VEL
LIN {X 0,Y 688.566,Z 200.105,A -85,B 0,C 180,E1 -3012.094,E2 -3012.094} C_VEL
LIN {X 0,Y 688.461,Z 199.476,A -85,B 0,C 180,E1 -3012.172,E2 -3012.172} C_VEL
LIN {X 0,Y 688.417,Z 199.481,A -85,B 0,C 180,E1 -3015.255,E2 -3015.255} C_VEL
LIN {X 0,Y 688.446,Z 199.477,A -85,B 0,C 180,E1 -3018.079,E2 -3018.079} C_VEL
LIN {X 0,Y 688.42,Z 199.481,A -85,B 0,C 180,E1 -3021.257,E2 -3021.257} C_VEL
LIN {X 0,Y 688.436,Z 199.53,A -85,B 0,C 180,E1 -3023.969,E2 -3023.969} C_VEL
LIN {X 0,Y 689.691,Z 202.873,A -85,B 0,C 180,E1 -3024.352,E2 -3024.352} C_VEL
LIN {X 0,Y 693.396,Z 211.165,A -85,B 0,C 180,E1 -3025.281,E2 -3025.281} C_VEL
LIN {X 0,Y 696.871,Z 220.343,A -85,B 0,C 180,E1 -3026.178,E2 -3026.178} C_VEL
LIN {X 0,Y 694.716,Z 266.624,A -85,B 0,C 180,E1 -3029.038,E2 -3029.038} C_VEL
LIN {X 0,Y 693.093,Z 322.938,A -85,B 0,C 180,E1 -3032.349,E2 -3032.349} C_VEL
LIN {X 0,Y 692.042,Z 375.961,A -85,B 0,C 180,E1 -3035.36,E2 -3035.36} C_VEL
LIN {X 0,Y 691.144,Z 430.671,A -85,B 0,C 180,E1 -3038.39,E2 -3038.39} C_VEL
LIN {X 0,Y 690.744,Z 462.706,A -85,B 0,C 180,E1 -3040.115,E2 -3040.115} C_VEL
LIN {X 0,Y 692.647,Z 479.634,A -85,B 0,C 180,E1 -3040.414,E2 -3040.414} C_VEL
LIN {X 0,Y 691.201,Z 622.884,A -85,B 0,C 180,E1 -3042.104,E2 -3042.104} C_VEL
LIN {X 0,Y 690.846,Z 681.611,A -85,B 0,C 180,E1 -3042.791,E2 -3042.791} C_VEL
LIN {X 0,Y 690.614,Z 700.894,A -85,B 0,C 180,E1 -3043.173,E2 -3043.173} C_VEL
LIN {X 0,Y 690.343,Z 718.904,A -85,B 0,C 180,E1 -3043.681,E2 -3043.681} C_VEL
LIN {X 0,Y 690.011,Z 736.238,A -85,B 0,C 180,E1 -3044.32,E2 -3044.32} C_VEL
LIN {X 0,Y 689.69,Z 752.449,A -85,B 0,C 180,E1 -3045.073,E2 -3045.073} C_VEL
LIN {X 0,Y 689.339,Z 768.367,A -85,B 0,C 180,E1 -3045.981,E2 -3045.981} C_VEL
LIN {X 0,Y 688.989,Z 783.057,A -85,B 0,C 180,E1 -3047,E2 -3047} C_VEL
LIN {X 0,Y 688.669,Z 796.479,A -85,B 0,C 180,E1 -3048.124,E2 -3048.124} C_VEL
LIN {X 0,Y 688.393,Z 808.805,A -85,B 0,C 180,E1 -3049.37,E2 -3049.37} C_VEL
LIN {X 0,Y 688.188,Z 820.655,A -85,B 0,C 180,E1 -3050.803,E2 -3050.803} C_VEL
LIN {X 0,Y 688.057,Z 830.244,A -85,B 0,C 180,E1 -3052.233,E2 -3052.233} C_VEL
LIN {X 0,Y 687.976,Z 837.865,A -85,B 0,C 180,E1 -3053.658,E2 -3053.658} C_VEL
LIN {X 0,Y 687.936,Z 844.054,A -85,B 0,C 180,E1 -3055.164,E2 -3055.164} C_VEL
LIN {X 0,Y 687.915,Z 848.471,A -85,B 0,C 180,E1 -3056.667,E2 -3056.667} C_VEL
LIN {X 0,Y 687.914,Z 851.344,A -85,B 0,C 180,E1 -3058.251,E2 -3058.251} C_VEL
LIN {X 0,Y 687.915,Z 852.449,A -85,B 0,C 180,E1 -3059.833,E2 -3059.833} C_VEL
LIN {X 0,Y 687.911,Z 851.815,A -85,B 0,C 180,E1 -3061.416,E2 -3061.416} C_VEL
LIN {X 0,Y 687.919,Z 849.427,A -85,B 0,C 180,E1 -3062.999,E2 -3062.999} C_VEL
LIN {X 0,Y 687.927,Z 845.478,A -85,B 0,C 180,E1 -3064.502,E2 -3064.502} C_VEL
LIN {X 0,Y 687.961,Z 839.805,A -85,B 0,C 180,E1 -3066.007,E2 -3066.007} C_VEL
LIN {X 0,Y 688.032,Z 832.71,A -85,B 0,C 180,E1 -3067.432,E2 -3067.432} C_VEL
LIN {X 0,Y 688.142,Z 823.731,A -85,B 0,C 180,E1 -3068.862,E2 -3068.862} C_VEL
LIN {X 0,Y 688.311,Z 813.319,A -85,B 0,C 180,E1 -3070.208,E2 -3070.208} C_VEL
LIN {X 0,Y 688.567,Z 800.725,A -85,B 0,C 180,E1 -3071.56,E2 -3071.56} C_VEL
LIN {X 0,Y 688.87,Z 787.333,A -85,B 0,C 180,E1 -3072.746,E2 -3072.746} C_VEL
LIN {X 0,Y 689.204,Z 772.853,A -85,B 0,C 180,E1 -3073.807,E2 -3073.807} C_VEL
LIN {X 0,Y 689.555,Z 757.405,A -85,B 0,C 180,E1 -3074.743,E2 -3074.743} C_VEL
LIN {X 0,Y 689.877,Z 741.064,A -85,B 0,C 180,E1 -3075.553,E2 -3075.553} C_VEL
LIN {X 0,Y 690.236,Z 723.857,A -85,B 0,C 180,E1 -3076.235,E2 -3076.235} C_VEL
LIN {X 0,Y 690.53,Z 705.346,A -85,B 0,C 180,E1 -3076.799,E2 -3076.799} C_VEL
LIN {X 0,Y 690.77,Z 686.648,A -85,B 0,C 180,E1 -3077.207,E2 -3077.207} C_VEL
LIN {X 0,Y 690.94,Z 665.223,A -85,B 0,C 180,E1 -3077.5,E2 -3077.5} C_VEL
LIN {X 0,Y 691.079,Z 629.682,A -85,B 0,C 180,E1 -3077.888,E2 -3077.888} C_VEL
LIN {X 0,Y 690.185,Z 622.078,A -85,B 0,C 180,E1 -3077.996,E2 -3077.996} C_VEL
LIN {X 0,Y 684.349,Z 602.175,A -85,B 0,C 180,E1 -3078.382,E2 -3078.382} C_VEL
LIN {X 0,Y 683.666,Z 595.646,A -85,B 0,C 180,E1 -3078.476,E2 -3078.476} C_VEL
LIN {X 0,Y 684.359,Z 477.101,A -85,B 0,C 180,E1 -3079.831,E2 -3079.831} C_VEL
LIN {X 0,Y 683.081,Z 466.178,A -85,B 0,C 180,E1 -3080.031,E2 -3080.031} C_VEL
LIN {X 0,Y 684.091,Z 410.724,A -85,B 0,C 180,E1 -3083.107,E2 -3083.107} C_VEL
LIN {X 0,Y 685.114,Z 357.611,A -85,B 0,C 180,E1 -3086.106,E2 -3086.106} C_VEL
LIN {X 0,Y 686.192,Z 308.344,A -85,B 0,C 180,E1 -3088.933,E2 -3088.933} C_VEL
LIN {X 0,Y 687.528,Z 254.78,A -85,B 0,C 180,E1 -3092.062,E2 -3092.062} C_VEL
LIN {X 0,Y 688.374,Z 221.597,A -85,B 0,C 180,E1 -3094.039,E2 -3094.039} C_VEL
LIN {X 0,Y 680.517,Z 200.457,A -85,B 0,C 180,E1 -3095.8,E2 -3095.8} C_VEL
LIN {X 0,Y 680.464,Z 200.468,A -85,B 0,C 180,E1 -3098.646,E2 -3098.646} C_VEL
LIN {X 0,Y 680.506,Z 200.466,A -85,B 0,C 180,E1 -3101.617,E2 -3101.617} C_VEL
LIN {X 0,Y 680.516,Z 200.465,A -85,B 0,C 180,E1 -3104.615,E2 -3104.615} C_VEL
LIN {X 0,Y 680.525,Z 200.46,A -85,B 0,C 180,E1 -3107.706,E2 -3107.706} C_VEL
LIN {X 0,Y 680.452,Z 200.467,A -85,B 0,C 180,E1 -3110.618,E2 -3110.618} C_VEL
LIN {X 0,Y 680.535,Z 200.535,A -85,B 0,C 180,E1 -3113.536,E2 -3113.536} C_VEL
LIN {X 0,Y 686.453,Z 215.886,A -85,B 0,C 180,E1 -3114.947,E2 -3114.947} C_VEL
LIN {X 0,Y 688.911,Z 223.653,A -85,B 0,C 180,E1 -3115.675,E2 -3115.675} C_VEL
LIN {X 0,Y 687.771,Z 263.046,A -85,B 0,C 180,E1 -3118.539,E2 -3118.539} C_VEL
LIN {X 0,Y 686.505,Z 299.257,A -85,B 0,C 180,E1 -3121.177,E2 -3121.177} C_VEL
LIN {X 0,Y 686.257,Z 307.834,A -85,B 0,C 180,E1 -3121.791,E2 -3121.791} C_VEL
LIN {X 0,Y 688.261,Z 319.043,A -85,B 0,C 180,E1 -3122.014,E2 -3122.014} C_VEL
LIN {X 0,Y 686.423,Z 604.169,A -85,B 0,C 180,E1 -3125.221,E2 -3125.221} C_VEL
LIN {X 0,Y 686.158,Z 621.906,A -85,B 0,C 180,E1 -3125.507,E2 -3125.507} C_VEL
LIN {X 0,Y 685.806,Z 639.574,A -85,B 0,C 180,E1 -3125.893,E2 -3125.893} C_VEL
LIN {X 0,Y 685.366,Z 656.998,A -85,B 0,C 180,E1 -3126.377,E2 -3126.377} C_VEL
LIN {X 0,Y 684.883,Z 675.569,A -85,B 0,C 180,E1 -3127.012,E2 -3127.012} C_VEL
LIN {X 0,Y 684.193,Z 697.588,A -85,B 0,C 180,E1 -3127.94,E2 -3127.94} C_VEL
LIN {X 0,Y 683.576,Z 715.679,A -85,B 0,C 180,E1 -3128.865,E2 -3128.865} C_VEL
LIN {X 0,Y 682.983,Z 731.983,A -85,B 0,C 180,E1 -3129.832,E2 -3129.832} C_VEL
LIN {X 0,Y 682.442,Z 747.427,A -85,B 0,C 180,E1 -3130.885,E2 -3130.885} C_VEL
LIN {X 0,Y 681.841,Z 764.705,A -85,B 0,C 180,E1 -3132.24,E2 -3132.24} C_VEL
LIN {X 0,Y 681.295,Z 780.672,A -85,B 0,C 180,E1 -3133.721,E2 -3133.721} C_VEL
LIN {X 0,Y 680.919,Z 793.306,A -85,B 0,C 180,E1 -3135.07,E2 -3135.07} C_VEL
LIN {X 0,Y 680.58,Z 805.591,A -85,B 0,C 180,E1 -3136.577,E2 -3136.577} C_VEL
LIN {X 0,Y 680.298,Z 817.976,A -85,B 0,C 180,E1 -3138.383,E2 -3138.383} C_VEL
LIN {X 0,Y 680.127,Z 827.25,A -85,B 0,C 180,E1 -3140.01,E2 -3140.01} C_VEL
LIN {X 0,Y 680.021,Z 835.299,A -85,B 0,C 180,E1 -3141.718,E2 -3141.718} C_VEL
LIN {X 0,Y 679.948,Z 842.269,A -85,B 0,C 180,E1 -3143.583,E2 -3143.583} C_VEL
LIN {X 0,Y 679.918,Z 847.307,A -85,B 0,C 180,E1 -3145.445,E2 -3145.445} C_VEL
LIN {X 0,Y 679.908,Z 850.487,A -85,B 0,C 180,E1 -3147.218,E2 -3147.218} C_VEL
LIN {X 0,Y 679.9,Z 852.132,A -85,B 0,C 180,E1 -3148.904,E2 -3148.904} C_VEL
LIN {X 0,Y 679.91,Z 852.329,A -85,B 0,C 180,E1 -3150.843,E2 -3150.843} C_VEL
LIN {X 0,Y 679.912,Z 850.73,A -85,B 0,C 180,E1 -3152.697,E2 -3152.697} C_VEL
LIN {X 0,Y 679.923,Z 847.849,A -85,B 0,C 180,E1 -3154.389,E2 -3154.389} C_VEL
LIN {X 0,Y 679.948,Z 843.297,A -85,B 0,C 180,E1 -3156.162,E2 -3156.162} C_VEL
LIN {X 0,Y 680.014,Z 836.027,A -85,B 0,C 180,E1 -3158.2,E2 -3158.2} C_VEL
LIN {X 0,Y 680.112,Z 828.15,A -85,B 0,C 180,E1 -3159.905,E2 -3159.905} C_VEL
LIN {X 0,Y 680.263,Z 819.549,A -85,B 0,C 180,E1 -3161.445,E2 -3161.445} C_VEL
LIN {X 0,Y 680.526,Z 808.194,A -85,B 0,C 180,E1 -3163.164,E2 -3163.164} C_VEL
LIN {X 0,Y 680.864,Z 795.192,A -85,B 0,C 180,E1 -3164.805,E2 -3164.805} C_VEL
LIN {X 0,Y 681.219,Z 783.264,A -85,B 0,C 180,E1 -3166.106,E2 -3166.106} C_VEL
LIN {X 0,Y 681.65,Z 770.12,A -85,B 0,C 180,E1 -3167.368,E2 -3167.368} C_VEL
LIN {X 0,Y 682.171,Z 755.037,A -85,B 0,C 180,E1 -3168.635,E2 -3168.635} C_VEL
LIN {X 0,Y 682.874,Z 735.446,A -85,B 0,C 180,E1 -3170.037,E2 -3170.037} C_VEL
LIN {X 0,Y 683.454,Z 718.898,A -85,B 0,C 180,E1 -3171.044,E2 -3171.044} C_VEL
LIN {X 0,Y 684.007,Z 702.968,A -85,B 0,C 180,E1 -3171.886,E2 -3171.886} C_VEL
LIN {X 0,Y 684.517,Z 686.647,A -85,B 0,C 180,E1 -3172.633,E2 -3172.633} C_VEL
LIN {X 0,Y 685.073,Z 668.594,A -85,B 0,C 180,E1 -3173.332,E2 -3173.332} C_VEL
LIN {X 0,Y 685.682,Z 646.288,A -85,B 0,C 180,E1 -3174.03,E2 -3174.03} C_VEL
LIN {X 0,Y 686.107,Z 624.882,A -85,B 0,C 180,E1 -3174.526,E2 -3174.526} C_VEL
LIN {X 0,Y 686.401,Z 606.327,A -85,B 0,C 180,E1 -3174.839,E2 -3174.839} C_VEL
LIN {X 0,Y 687.07,Z 504.663,A -85,B 0,C 180,E1 -3175.991,E2 -3175.991} C_VEL
LIN {X 0,Y 688.092,Z 316.943,A -85,B 0,C 180,E1 -3178.108,E2 -3178.108} C_VEL
LIN {X 0,Y 686.181,Z 307.3,A -85,B 0,C 180,E1 -3178.315,E2 -3178.315} C_VEL
LIN {X 0,Y 687.433,Z 274.484,A -85,B 0,C 180,E1 -3180.725,E2 -3180.725} C_VEL
LIN {X 0,Y 688.659,Z 233.526,A -85,B 0,C 180,E1 -3183.699,E2 -3183.699} C_VEL
LIN {X 0,Y 688.736,Z 222.447,A -85,B 0,C 180,E1 -3184.517,E2 -3184.517} C_VEL
LIN {X 0,Y 682.873,Z 206.786,A -85,B 0,C 180,E1 -3186.002,E2 -3186.002} C_VEL
LIN {X 0,Y 680.513,Z 200.463,A -85,B 0,C 180,E1 -3186.565,E2 -3186.565} C_VEL
LIN {X 0,Y 680.524,Z 200.466,A -85,B 0,C 180,E1 -3189.654,E2 -3189.654} C_VEL
LIN {X 0,Y 680.504,Z 200.461,A -85,B 0,C 180,E1 -3192.753,E2 -3192.753} C_VEL
LIN {X 0,Y 680.522,Z 200.462,A -85,B 0,C 180,E1 -3195.74,E2 -3195.74} C_VEL
LIN {X 0,Y 680.505,Z 200.46,A -85,B 0,C 180,E1 -3198.832,E2 -3198.832} C_VEL
LIN {X 0,Y 680.522,Z 200.463,A -85,B 0,C 180,E1 -3201.82,E2 -3201.82} C_VEL
LIN {X 0,Y 680.505,Z 200.459,A -85,B 0,C 180,E1 -3204.927,E2 -3204.927} C_VEL
LIN {X 0,Y 680.52,Z 200.461,A -85,B 0,C 180,E1 -3207.867,E2 -3207.867} C_VEL
LIN {X 0,Y 680.511,Z 200.453,A -85,B 0,C 180,E1 -3210.899,E2 -3210.899} C_VEL
LIN {X 0,Y 680.516,Z 200.463,A -85,B 0,C 180,E1 -3213.939,E2 -3213.939} C_VEL
LIN {X 0,Y 680.511,Z 200.447,A -85,B 0,C 180,E1 -3216.993,E2 -3216.993} C_VEL
LIN {X 0,Y 680.513,Z 200.459,A -85,B 0,C 180,E1 -3219.98,E2 -3219.98} C_VEL
LIN {X 0,Y 680.513,Z 200.45,A -85,B 0,C 180,E1 -3223.043,E2 -3223.043} C_VEL
LIN {X 0,Y 680.508,Z 200.457,A -85,B 0,C 180,E1 -3226.056,E2 -3226.056} C_VEL
LIN {X 0,Y 680.517,Z 200.45,A -85,B 0,C 180,E1 -3229.074,E2 -3229.074} C_VEL
LIN {X 0,Y 680.507,Z 200.459,A -85,B 0,C 180,E1 -3232.061,E2 -3232.061} C_VEL
LIN {X 0,Y 680.518,Z 200.448,A -85,B 0,C 180,E1 -3235.111,E2 -3235.111} C_VEL
LIN {X 0,Y 680.503,Z 200.46,A -85,B 0,C 180,E1 -3238.148,E2 -3238.148} C_VEL
LIN {X 0,Y 680.523,Z 200.443,A -85,B 0,C 180,E1 -3241.094,E2 -3241.094} C_VEL
LIN {X 0,Y 680.503,Z 200.463,A -85,B 0,C 180,E1 -3244.129,E2 -3244.129} C_VEL
LIN {X 0,Y 680.524,Z 200.444,A -85,B 0,C 180,E1 -3247.174,E2 -3247.174} C_VEL
LIN {X 0,Y 680.496,Z 200.463,A -85,B 0,C 180,E1 -3250.241,E2 -3250.241} C_VEL
LIN {X 0,Y 680.525,Z 200.456,A -85,B 0,C 180,E1 -3253.251,E2 -3253.251} C_VEL
LIN {X 0,Y 680.489,Z 200.464,A -85,B 0,C 180,E1 -3256.299,E2 -3256.299} C_VEL
LIN {X 0,Y 680.522,Z 200.455,A -85,B 0,C 180,E1 -3259.216,E2 -3259.216} C_VEL
LIN {X 0,Y 680.49,Z 200.465,A -85,B 0,C 180,E1 -3262.278,E2 -3262.278} C_VEL
LIN {X 0,Y 680.518,Z 200.457,A -85,B 0,C 180,E1 -3265.22,E2 -3265.22} C_VEL
LIN {X 0,Y 680.485,Z 200.464,A -85,B 0,C 180,E1 -3268.339,E2 -3268.339} C_VEL
LIN {X 0,Y 680.516,Z 200.458,A -85,B 0,C 180,E1 -3271.243,E2 -3271.243} C_VEL
LIN {X 0,Y 680.483,Z 200.466,A -85,B 0,C 180,E1 -3274.35,E2 -3274.35} C_VEL
LIN {X 0,Y 680.507,Z 200.46,A -85,B 0,C 180,E1 -3277.255,E2 -3277.255} C_VEL
LIN {X 0,Y 680.486,Z 200.468,A -85,B 0,C 180,E1 -3280.306,E2 -3280.306} C_VEL
LIN {X 0,Y 680.484,Z 200.463,A -85,B 0,C 180,E1 -3283.099,E2 -3283.099} C_VEL
LIN {X 0,Y 680.497,Z 200.468,A -85,B 0,C 180,E1 -3286.206,E2 -3286.206} C_VEL
LIN {X 0,Y 680.546,Z 200.608,A -85,B 0,C 180,E1 -3287.649,E2 -3287.649} C_VEL
LIN {X 0,Y 681.71,Z 203.762,A -85,B 0,C 180,E1 -3287.917,E2 -3287.917} C_VEL
LIN {X 0,Y 689.851,Z 220.391,A -85,B 0,C 180,E1 -3289.421,E2 -3289.421} C_VEL
LIN {X 0,Y 693.4,Z 228.06,A -85,B 0,C 180,E1 -3290.055,E2 -3290.055} C_VEL
LIN {X 0,Y 691.864,Z 284.655,A -85,B 0,C 180,E1 -3292.78,E2 -3292.78} C_VEL
LIN {X 0,Y 691.551,Z 300.07,A -85,B 0,C 180,E1 -3293.489,E2 -3293.489} C_VEL
LIN {X 0,Y 693.628,Z 313.843,A -85,B 0,C 180,E1 -3293.764,E2 -3293.764} C_VEL
LIN {X 0,Y 691.532,Z 571.069,A -85,B 0,C 180,E1 -3296.81,E2 -3296.81} C_VEL
LIN {X 0,Y 690.512,Z 691.443,A -85,B 0,C 180,E1 -3298.236,E2 -3298.236} C_VEL
LIN {X 0,Y 689.975,Z 716.757,A -85,B 0,C 180,E1 -3298.684,E2 -3298.684} C_VEL
LIN {X 0,Y 689.34,Z 738.451,A -85,B 0,C 180,E1 -3299.204,E2 -3299.204} C_VEL
LIN {X 0,Y 688.601,Z 762.554,A -85,B 0,C 180,E1 -3299.936,E2 -3299.936} C_VEL
LIN {X 0,Y 687.791,Z 783.606,A -85,B 0,C 180,E1 -3300.723,E2 -3300.723} C_VEL
LIN {X 0,Y 686.892,Z 805.964,A -85,B 0,C 180,E1 -3301.704,E2 -3301.704} C_VEL
LIN {X 0,Y 685.951,Z 827.052,A -85,B 0,C 180,E1 -3302.803,E2 -3302.803} C_VEL
LIN {X 0,Y 685.062,Z 846.93,A -85,B 0,C 180,E1 -3303.987,E2 -3303.987} C_VEL
LIN {X 0,Y 684.091,Z 867.293,A -85,B 0,C 180,E1 -3305.387,E2 -3305.387} C_VEL
LIN {X 0,Y 683.28,Z 885.609,A -85,B 0,C 180,E1 -3306.818,E2 -3306.818} C_VEL
LIN {X 0,Y 682.485,Z 903.534,A -85,B 0,C 180,E1 -3308.424,E2 -3308.424} C_VEL
LIN {X 0,Y 681.84,Z 919.628,A -85,B 0,C 180,E1 -3310.052,E2 -3310.052} C_VEL
LIN {X 0,Y 681.28,Z 934.522,A -85,B 0,C 180,E1 -3311.783,E2 -3311.783} C_VEL
LIN {X 0,Y 680.844,Z 947.817,A -85,B 0,C 180,E1 -3313.537,E2 -3313.537} C_VEL
LIN {X 0,Y 680.499,Z 960.282,A -85,B 0,C 180,E1 -3315.448,E2 -3315.448} C_VEL
LIN {X 0,Y 680.267,Z 970.026,A -85,B 0,C 180,E1 -3317.177,E2 -3317.177} C_VEL
LIN {X 0,Y 680.079,Z 979.831,A -85,B 0,C 180,E1 -3319.238,E2 -3319.238} C_VEL
LIN {X 0,Y 679.975,Z 986.817,A -85,B 0,C 180,E1 -3321.033,E2 -3321.033} C_VEL
LIN {X 0,Y 679.949,Z 993.141,A -85,B 0,C 180,E1 -3323.034,E2 -3323.034} C_VEL
LIN {X 0,Y 679.895,Z 997.657,A -85,B 0,C 180,E1 -3325.022,E2 -3325.022} C_VEL
LIN {X 0,Y 679.893,Z 1000.462,A -85,B 0,C 180,E1 -3326.796,E2 -3326.796} C_VEL
LIN {X 0,Y 679.908,Z 1002.216,A -85,B 0,C 180,E1 -3328.905,E2 -3328.905} C_VEL
LIN {X 0,Y 679.883,Z 1002.328,A -85,B 0,C 180,E1 -3330.674,E2 -3330.674} C_VEL
LIN {X 0,Y 679.895,Z 1001.227,A -85,B 0,C 180,E1 -3332.529,E2 -3332.529} C_VEL
LIN {X 0,Y 679.916,Z 998.29,A -85,B 0,C 180,E1 -3334.639,E2 -3334.639} C_VEL
LIN {X 0,Y 679.923,Z 994.483,A -85,B 0,C 180,E1 -3336.417,E2 -3336.417} C_VEL
LIN {X 0,Y 679.965,Z 988.635,A -85,B 0,C 180,E1 -3338.456,E2 -3338.456} C_VEL
LIN {X 0,Y 680.074,Z 981.384,A -85,B 0,C 180,E1 -3340.387,E2 -3340.387} C_VEL
LIN {X 0,Y 680.222,Z 972.709,A -85,B 0,C 180,E1 -3342.307,E2 -3342.307} C_VEL
LIN {X 0,Y 680.456,Z 961.84,A -85,B 0,C 180,E1 -3344.292,E2 -3344.292} C_VEL
LIN {X 0,Y 680.777,Z 950.047,A -85,B 0,C 180,E1 -3346.144,E2 -3346.144} C_VEL
LIN {X 0,Y 681.229,Z 935.929,A -85,B 0,C 180,E1 -3348.041,E2 -3348.041} C_VEL
LIN {X 0,Y 681.78,Z 920.971,A -85,B 0,C 180,E1 -3349.803,E2 -3349.803} C_VEL
LIN {X 0,Y 682.449,Z 904.46,A -85,B 0,C 180,E1 -3351.487,E2 -3351.487} C_VEL
LIN {X 0,Y 683.235,Z 886.712,A -85,B 0,C 180,E1 -3353.092,E2 -3353.092} C_VEL
LIN {X 0,Y 684.071,Z 867.771,A -85,B 0,C 180,E1 -3354.577,E2 -3354.577} C_VEL
LIN {X 0,Y 685.031,Z 847.628,A -85,B 0,C 180,E1 -3355.969,E2 -3355.969} C_VEL
LIN {X 0,Y 685.913,Z 827.937,A -85,B 0,C 180,E1 -3357.147,E2 -3357.147} C_VEL
LIN {X 0,Y 686.869,Z 806.495,A -85,B 0,C 180,E1 -3358.271,E2 -3358.271} C_VEL
LIN {X 0,Y 687.759,Z 784.48,A -85,B 0,C 180,E1 -3359.241,E2 -3359.241} C_VEL
LIN {X 0,Y 688.548,Z 763.835,A -85,B 0,C 180,E1 -3360.018,E2 -3360.018} C_VEL
LIN {X 0,Y 689.331,Z 738.773,A -85,B 0,C 180,E1 -3360.787,E2 -3360.787} C_VEL
LIN {X 0,Y 689.962,Z 717.146,A -85,B 0,C 180,E1 -3361.307,E2 -3361.307} C_VEL
LIN {X 0,Y 690.509,Z 691.704,A -85,B 0,C 180,E1 -3361.76,E2 -3361.76} C_VEL
LIN {X 0,Y 691.408,Z 586.497,A -85,B 0,C 180,E1 -3363.009,E2 -3363.009} C_VEL
LIN {X 0,Y 693.602,Z 318.417,A -85,B 0,C 180,E1 -3366.183,E2 -3366.183} C_VEL
LIN {X 0,Y 693.37,Z 310.96,A -85,B 0,C 180,E1 -3366.281,E2 -3366.281} C_VEL
LIN {X 0,Y 691.268,Z 298.667,A -85,B 0,C 180,E1 -3366.528,E2 -3366.528} C_VEL
LIN {X 0,Y 691.963,Z 260.145,A -85,B 0,C 180,E1 -3368.312,E2 -3368.312} C_VEL
LIN {X 0,Y 693.257,Z 227.855,A -85,B 0,C 180,E1 -3369.928,E2 -3369.928} C_VEL
LIN {X 0,Y 686.717,Z 213.41,A -85,B 0,C 180,E1 -3371.326,E2 -3371.326} C_VEL
LIN {X 0,Y 682.333,Z 204.616,A -85,B 0,C 180,E1 -3372.391,E2 -3372.391} C_VEL
LIN {X 0,Y 680.649,Z 201.213,A -85,B 0,C 180,E1 -3372.857,E2 -3372.857} C_VEL
LIN {X 0,Y 680.521,Z 200.466,A -85,B 0,C 180,E1 -3372.981,E2 -3372.981} C_VEL
LIN {X 0,Y 680.507,Z 200.467,A -85,B 0,C 180,E1 -3375.973,E2 -3375.973} C_VEL
LIN {X 0,Y 680.523,Z 200.466,A -85,B 0,C 180,E1 -3379.045,E2 -3379.045} C_VEL
LIN {X 0,Y 680.524,Z 200.466,A -85,B 0,C 180,E1 -3382.109,E2 -3382.109} C_VEL
LIN {X 0,Y 680.554,Z 200.698,A -85,B 0,C 180,E1 -3383.26,E2 -3383.26} C_VEL
LIN {X 0,Y 682.051,Z 204.299,A -85,B 0,C 180,E1 -3383.736,E2 -3383.736} C_VEL
LIN {X 0,Y 685.777,Z 212.313,A -85,B 0,C 180,E1 -3384.736,E2 -3384.736} C_VEL
LIN {X 0,Y 690.176,Z 223.8,A -85,B 0,C 180,E1 -3385.934,E2 -3385.934} C_VEL
LIN {X 0,Y 687.73,Z 268.398,A -85,B 0,C 180,E1 -3388.748,E2 -3388.748} C_VEL
LIN {X 0,Y 685.83,Z 323.875,A -85,B 0,C 180,E1 -3392.068,E2 -3392.068} C_VEL
LIN {X 0,Y 684.59,Z 376.896,A -85,B 0,C 180,E1 -3395.125,E2 -3395.125} C_VEL
LIN {X 0,Y 683.539,Z 431.477,A -85,B 0,C 180,E1 -3398.188,E2 -3398.188} C_VEL
LIN {X 0,Y 683.134,Z 459.994,A -85,B 0,C 180,E1 -3399.744,E2 -3399.744} C_VEL
LIN {X 0,Y 685.436,Z 480.384,A -85,B 0,C 180,E1 -3400.131,E2 -3400.131} C_VEL
LIN {X 0,Y 683.692,Z 621.003,A -85,B 0,C 180,E1 -3401.854,E2 -3401.854} C_VEL
LIN {X 0,Y 683.238,Z 681.836,A -85,B 0,C 180,E1 -3402.586,E2 -3402.586} C_VEL
LIN {X 0,Y 682.981,Z 701.179,A -85,B 0,C 180,E1 -3402.974,E2 -3402.974} C_VEL
LIN {X 0,Y 682.68,Z 719.393,A -85,B 0,C 180,E1 -3403.492,E2 -3403.492} C_VEL
LIN {X 0,Y 682.322,Z 736.765,A -85,B 0,C 180,E1 -3404.139,E2 -3404.139} C_VEL
LIN {X 0,Y 681.971,Z 752.982,A -85,B 0,C 180,E1 -3404.897,E2 -3404.897} C_VEL
LIN {X 0,Y 681.609,Z 768.373,A -85,B 0,C 180,E1 -3405.776,E2 -3405.776} C_VEL
LIN {X 0,Y 681.227,Z 783.257,A -85,B 0,C 180,E1 -3406.806,E2 -3406.806} C_VEL
LIN {X 0,Y 680.897,Z 796.161,A -85,B 0,C 180,E1 -3407.878,E2 -3407.878} C_VEL
LIN {X 0,Y 680.603,Z 808.196,A -85,B 0,C 180,E1 -3409.075,E2 -3409.075} C_VEL
LIN {X 0,Y 680.352,Z 818.873,A -85,B 0,C 180,E1 -3410.355,E2 -3410.355} C_VEL
LIN {X 0,Y 680.158,Z 828.192,A -85,B 0,C 180,E1 -3411.717,E2 -3411.717} C_VEL
LIN {X 0,Y 680.025,Z 836.118,A -85,B 0,C 180,E1 -3413.16,E2 -3413.16} C_VEL
LIN {X 0,Y 679.955,Z 842.584,A -85,B 0,C 180,E1 -3414.684,E2 -3414.684} C_VEL
LIN {X 0,Y 679.922,Z 847.646,A -85,B 0,C 180,E1 -3416.29,E2 -3416.29} C_VEL
LIN {X 0,Y 679.911,Z 850.776,A -85,B 0,C 180,E1 -3417.809,E2 -3417.809} C_VEL
LIN {X 0,Y 679.915,Z 852.336,A -85,B 0,C 180,E1 -3419.41,E2 -3419.41} C_VEL
LIN {X 0,Y 679.918,Z 852.154,A -85,B 0,C 180,E1 -3421.011,E2 -3421.011} C_VEL
LIN {X 0,Y 679.916,Z 850.224,A -85,B 0,C 180,E1 -3422.613,E2 -3422.613} C_VEL
LIN {X 0,Y 679.922,Z 846.748,A -85,B 0,C 180,E1 -3424.132,E2 -3424.132} C_VEL
LIN {X 0,Y 679.958,Z 841.259,A -85,B 0,C 180,E1 -3425.739,E2 -3425.739} C_VEL
LIN {X 0,Y 680.045,Z 834.309,A -85,B 0,C 180,E1 -3427.264,E2 -3427.264} C_VEL
LIN {X 0,Y 680.178,Z 825.862,A -85,B 0,C 180,E1 -3428.709,E2 -3428.709} C_VEL
LIN {X 0,Y 680.396,Z 815.288,A -85,B 0,C 180,E1 -3430.157,E2 -3430.157} C_VEL
LIN {X 0,Y 680.654,Z 803.831,A -85,B 0,C 180,E1 -3431.439,E2 -3431.439} C_VEL
LIN {X 0,Y 680.984,Z 790.402,A -85,B 0,C 180,E1 -3432.68,E2 -3432.68} C_VEL
LIN {X 0,Y 681.352,Z 775.779,A -85,B 0,C 180,E1 -3433.796,E2 -3433.796} C_VEL
LIN {X 0,Y 681.746,Z 760.057,A -85,B 0,C 180,E1 -3434.785,E2 -3434.785} C_VEL
LIN {X 0,Y 682.118,Z 743.276,A -85,B 0,C 180,E1 -3435.648,E2 -3435.648} C_VEL
LIN {X 0,Y 682.53,Z 725.39,A -85,B 0,C 180,E1 -3436.38,E2 -3436.38} C_VEL
LIN {X 0,Y 682.868,Z 706.517,A -85,B 0,C 180,E1 -3436.971,E2 -3436.971} C_VEL
LIN {X 0,Y 683.139,Z 687.496,A -85,B 0,C 180,E1 -3437.398,E2 -3437.398} C_VEL
LIN {X 0,Y 683.329,Z 666.69,A -85,B 0,C 180,E1 -3437.692,E2 -3437.692} C_VEL
LIN {X 0,Y 683.666,Z 595.646,A -85,B 0,C 180,E1 -3438.476,E2 -3438.476} C_VEL
LIN {X 0,Y 682.791,Z 588.053,A -85,B 0,C 180,E1 -3438.592,E2 -3438.592} C_VEL
LIN {X 0,Y 677.088,Z 568.181,A -85,B 0,C 180,E1 -3439.006,E2 -3439.006} C_VEL
LIN {X 0,Y 676.454,Z 561.656,A -85,B 0,C 180,E1 -3439.105,E2 -3439.105} C_VEL
LIN {X 0,Y 676.947,Z 477.791,A -85,B 0,C 180,E1 -3440.086,E2 -3440.086} C_VEL
LIN {X 0,Y 675.482,Z 465.394,A -85,B 0,C 180,E1 -3440.311,E2 -3440.311} C_VEL
LIN {X 0,Y 676.601,Z 409.918,A -85,B 0,C 180,E1 -3443.424,E2 -3443.424} C_VEL
LIN {X 0,Y 677.746,Z 356.691,A -85,B 0,C 180,E1 -3446.458,E2 -3446.458} C_VEL
LIN {X 0,Y 679.018,Z 304.926,A -85,B 0,C 180,E1 -3449.461,E2 -3449.461} C_VEL
LIN {X 0,Y 680.442,Z 252.93,A -85,B 0,C 180,E1 -3452.536,E2 -3452.536} C_VEL
LIN {X 0,Y 681.13,Z 224.316,A -85,B 0,C 180,E1 -3454.261,E2 -3454.261} C_VEL
LIN {X 0,Y 672.579,Z 201.441,A -85,B 0,C 180,E1 -3456.195,E2 -3456.195} C_VEL
LIN {X 0,Y 672.545,Z 201.456,A -85,B 0,C 180,E1 -3459.098,E2 -3459.098} C_VEL
LIN {X 0,Y 672.529,Z 201.456,A -85,B 0,C 180,E1 -3462.108,E2 -3462.108} C_VEL
LIN {X 0,Y 672.582,Z 201.45,A -85,B 0,C 180,E1 -3464.956,E2 -3464.956} C_VEL
LIN {X 0,Y 672.588,Z 201.453,A -85,B 0,C 180,E1 -3468.015,E2 -3468.015} C_VEL
LIN {X 0,Y 672.513,Z 201.456,A -85,B 0,C 180,E1 -3470.81,E2 -3470.81} C_VEL
